// Write Own Data to CIP
      L     DB1225.DBD   10;
      T     DB1225.DBD  154;

      L     DB1225.DBW   14;
      T     DB1225.DBW  158;

      L     DB1225.DBW   16;
      T     DB1225.DBW  160;

      L     DB1225.DBW   18;
      T     DB1225.DBW  162;

      L     DB1225.DBW   20;
      T     DB1225.DBW  164;

      L     DB1225.DBW   22;
      T     DB1225.DBW  166;

      A     DB1225.DBX   24.0;
      =     DB1225.DBX  168.0;

      A     DB1225.DBX   24.1;
      =     DB1225.DBX  168.1;

      A     DB1225.DBX   24.2;
      =     DB1225.DBX  168.2;

      A     DB1225.DBX   24.3;
      =     DB1225.DBX  168.3;

      A     DB1225.DBX   24.4;
      =     DB1225.DBX  168.4;

      A     DB1225.DBX   24.5;
      =     DB1225.DBX  168.5;

      A     DB1225.DBX   24.6;
      =     DB1225.DBX  168.6;

      A     DB1225.DBX   24.7;
      =     DB1225.DBX  168.7;

// Copy Data to CIP
      CALL SFC   20 (
           SRCBLK                   := DB1225.ToCIP,
           RET_VAL                  := #iRetVal,
           DSTBLK                   := DB1225.ToCIP);

NCIP: NOP   0;

//Empty Signal
//A     "U022SpID".SpI.Sig //!!!! Insert correct Empty Signal !!!
      CLR   ;
      =     DB1225.DBX   26.5;

//Full Signal
//A     "U022SpID".SpI.Sig //!!!! Insert correct Full Signal !!!
      CLR   ;
      =     DB1225.DBX   26.2;

//CIP Program Selected
      A     #CIP;
      =     DB1225.DBX   27.1;

// Emergency Stop
      A     #EStopOK; //If needed add or replace with own SpI
      =     DB1225.DBX   27.0; //Emergency Stop OK


NETWORK
TITLE = read from other unit data



END_FUNCTION_BLOCK

FUNCTION_BLOCK FB 1229
TITLE =U022: Well Transfer VE2
AUTHOR : Woermann
FAMILY : BOTEC_F1
NAME : Sim
VERSION : 0.1


VAR_TEMP
  CIP : BOOL ;	//CIP active
  xTmp : BOOL ;	//Temporary BOOL (free for general use)
  iTmp : INT ;	//Temporary INT (free for general use)
  rTmp : REAL ;	//Temporary REAL (free for general use)
  UnitNo : INT ;	//Unit Number
END_VAR
BEGIN
NETWORK
TITLE =General

      SET   ;
// get unit number ----------------------------------------------------------
      L     DB1220.DBW    0;
      T     #UnitNo;

// CIP ----------------------------------------------------------------------
      L     DB1221.DBD   54;
      L     0;
      <D    ;
      =     #CIP;

NETWORK
TITLE =Actuator

      A     DB1221.DBX   17.3;
      =     DB2220.DBX  105.3;
      =     DB2220.DBX  185.3;
      =     DB2220.DBX  265.3;

NETWORK
TITLE =Special Input

      A     DB1221.DBX   17.3;
      =     DB2221.DBX   81.3;
      =     DB2221.DBX  141.3;
      =     DB2221.DBX  201.3;

NETWORK
TITLE =Counter

      A     DB1221.DBX   17.3;
      A     M    101.0;


      CLR   ;
NETWORK
TITLE =Analog Input

      A     DB1221.DBX   17.3;
      =     DB2223.DBX  141.3;
      =     DB2223.DBX  261.3;
      =     DB2223.DBX  381.3;

NETWORK
TITLE =Universal Value

      A     DB1221.DBX   17.3;
//      =     "U022UnVD".unv001.Sim;
//      =     "U022UnVD".unv002.Sim;
//      =     "U022UnVD".unv003.Sim;
//      =     "U022UnVD".unv004.Sim;

NETWORK
TITLE =PID

      A     DB1221.DBX   17.3;
//      =     "U022PIDD".U22_PID001.Ign;

NETWORK
TITLE =Message

      A     DB1221.DBX   17.3;
//      =     "U022MsgD".msg001.Sim;
//      =     "U022MsgD".msg002.Sim;
//      =     "U022MsgD".msg003.Sim;

NETWORK
TITLE =VLT

      A     DB1221.DBX   17.3;

END_FUNCTION_BLOCK

FUNCTION_BLOCK FB 1255
TITLE =U025: Well Transfer A
FAMILY : BOTEC_F1
NAME : Comm
VERSION : 0.1


VAR_TEMP
  iRetVal : INT ;	//return value as integer
  wRetVal : WORD ;	//return value as word
  Run : BOOL ;	//Unit in "RUN" mode
  EStopOK : BOOL ;	//Emergency Stop OK
  CIP : BOOL ;	//CIP Program Selected
  ComCIP : BOOL ;	//Communication with CIP Active
  xTmp : BOOL ;	//Temporary BOOL (free for general use)
  iTmp : INT ;	//Temporary INT (free for general use)
  rTmp : REAL ;	//Temporary REAL (free for general use)
  dTmp : DINT ;	//Temporary DINT (free for general use)
  UnitNo : INT ;	//Unit Number
  EquipmentID : INT ;	//Equipment ID
  Prid : DINT ;	//Process ID
  SFM36 : STRUCT 	// CIP Pump Mode
   I00 : BOOL ;	// Off
   I01 : BOOL ;	// Flow
   I02 : BOOL ;	// Pressure
   I03 : BOOL ;	// Fix Speed
   I04 : BOOL ;
   I05 : BOOL ;
   I06 : BOOL ;
   I07 : BOOL ;
   I08 : BOOL ;
   I09 : BOOL ;
   I10 : BOOL ;
   I11 : BOOL ;
   I12 : BOOL ;
   I13 : BOOL ;
   I14 : BOOL ;
   I15 : BOOL ;
   I16 : BOOL ;
   I17 : BOOL ;
   I18 : BOOL ;
   I19 : BOOL ;
   I20 : BOOL ;
   I21 : BOOL ;
   I22 : BOOL ;
   I23 : BOOL ;
   I24 : BOOL ;
   I25 : BOOL ;
   I26 : BOOL ;
   I27 : BOOL ;
   I28 : BOOL ;
   I29 : BOOL ;
   I30 : BOOL ;
   I31 : BOOL ;
  END_STRUCT ;
END_VAR
BEGIN
NETWORK
TITLE =general

      SET   ;

// unit & equipment number ---------------------------------------------------
      L     DB1250.DBW    0;
      T     #UnitNo;

      L     DB1255.DBW   14;
      L     1000;
      *I    ;
      L     #UnitNo;
      +I    ;
      T     #EquipmentID;

// CIP ----------------------------------------------------------------------
      L     DB1255.DBW   18;
      L     0;
      <I    ;
      =     #CIP;

// Communicating Units-------------------------------------------------------
      L     DB1255.DBD   10;
      L     DB1255.DBD  106;
      ==D   ;
      =     #ComCIP;

// emergency OK -------------------------------------------------------------
      A     DB1255.DBX   75.0; //General Emergency Stop OK
      =     #EStopOK;

NETWORK
TITLE =read other unit's data

      SET   ;

// ... General Unit ----------/

      CALL FC   563 (
           ActReq                   := M    101.0,
           PLCNo                    := DB1255.DBW   14,
           SourceUnitNo             := 99,
           IsTUnit                  := FALSE,
           DstComDRec               := DB1255.GEN,
           RET_VAL                  := #wRetVal);


NETWORK
TITLE =remote start

      SET   ;
// !!! insert correct condition of unit start !!!
      A     DB1251.DBX   15.0;
      A     DB1251.DBX   17.4;
      CLR   ;
      JCN   Strt;
      L     DB1255.DBD   10;
//L        L#-1;                            // Prid negative to start on its own
      T     #Prid;

      CALL FC    48 (
           UnitNo                   := #UnitNo,
           PrId                     := #Prid,
           Run                      := DB1251.DBX   17.4,
           PrIdTransfer             := TRUE,
           Start                    := TRUE,
           RetVal                   := #wRetVal);
Strt: NOP   0;
NETWORK
TITLE =external releases

      SET   ;
      =     DB2250.DBX  106.7;
      =     DB2250.DBX  186.7;
      =     DB2250.DBX  266.7;
NETWORK
TITLE =write own unit data

      SET   ;

//-- CIP Communication ---------------------------------------
      AN    DB1251.DBX   15.0;
//      AN "U025SeqD".Seq.PO.B30 // CIP Active (Slave)
      A     #ComCIP;
      JCN   NCIP;
//Conductivity CIP Return
      L     DB1255.DBD  150;
      T     DB1251.DBD  626;

//Temperature CIP Return
      L     DB1255.DBD  146;
      T     DB1251.DBD  594;

//CIP Prerun Pump SP

      CALL FC    45 (
           SFM                      := DB1251.DBD  686,
           Indexes                  := #SFM36);


      L     0.000000e+000;
      A     #SFM36.I01;
      =     DB1255.DBX  171.7;
      JCN   pfc;
      L     DB1251.DBD  654;
pfc:  NOP   0;
      A     #SFM36.I02;
      =     DB1255.DBX  172.0;
      JCN   ppc;
      L     DB1251.DBD  670;
ppc:  NOP   0;
      A     #SFM36.I03;
      =     DB1255.DBX  171.6;
      JCN   pxc;
      L     DB1251.DBD  574;
pxc:  NOP   0;
      T     DB1255.DBD  182;

//CIP Return
      L     DB1251.DBD  558;
      T     DB1255.DBD  186;
      L     DB1255.DBD  138;
      T     DB1251.DBD  562;

//CIP Prerun
      L     DB1251.DBD  542;
      T     DB1255.DBD  190;
      L     DB1255.DBD  142;
      T     DB1251.DBD  546;

// Write Own Data to CIP
      L     DB1255.DBD   10;
      T     DB1255.DBD  154;

      L     DB1255.DBW   14;
      T     DB1255.DBW  158;

      L     DB1255.DBW   16;
      T     DB1255.DBW  160;

      L     DB1255.DBW   18;
      T     DB1255.DBW  162;

      L     DB1255.DBW   20;
      T     DB1255.DBW  164;

      L     DB1255.DBW   22;
      T     DB1255.DBW  166;

      A     DB1255.DBX   24.0;
      =     DB1255.DBX  168.0;

      A     DB1255.DBX   24.1;
      =     DB1255.DBX  168.1;

      A     DB1255.DBX   24.2;
      =     DB1255.DBX  168.2;

      A     DB1255.DBX   24.3;
      =     DB1255.DBX  168.3;

      A     DB1255.DBX   24.4;
      =     DB1255.DBX  168.4;

      A     DB1255.DBX   24.5;
      =     DB1255.DBX  168.5;

      A     DB1255.DBX   24.6;
      =     DB1255.DBX  168.6;

      A     DB1255.DBX   24.7;
      =     DB1255.DBX  168.7;

// Copy Data to CIP
      CALL SFC   20 (
           SRCBLK                   := DB1255.ToCIP,
           RET_VAL                  := #iRetVal,
           DSTBLK                   := DB1255.ToCIP);

NCIP: NOP   0;

//Empty Signal
//A     "U025SpID".SpI.Sig //!!!! Insert correct Empty Signal !!!
      CLR   ;
      =     DB1255.DBX   26.5;

//Full Signal
//A     "U025SpID".SpI.Sig //!!!! Insert correct Full Signal !!!
      CLR   ;
      =     DB1255.DBX   26.2;

//CIP Program Selected
      A     #CIP;
      =     DB1255.DBX   27.1;

// Emergency Stop
      A     #EStopOK; //If needed add or replace with own SpI
      =     DB1255.DBX   27.0; //Emergency Stop OK


NETWORK
TITLE = read from other unit data



END_FUNCTION_BLOCK

FUNCTION_BLOCK FB 1259
TITLE =U025: Well Transfer A
AUTHOR : Woermann
FAMILY : BOTEC_F1
NAME : Sim
VERSION : 0.1


VAR_TEMP
  CIP : BOOL ;	//CIP active
  xTmp : BOOL ;	//Temporary BOOL (free for general use)
  iTmp : INT ;	//Temporary INT (free for general use)
  rTmp : REAL ;	//Temporary REAL (free for general use)
  UnitNo : INT ;	//Unit Number
END_VAR
BEGIN
NETWORK
TITLE =General

      SET   ;
// get unit number ----------------------------------------------------------
      L     DB1250.DBW    0;
      T     #UnitNo;

// CIP ----------------------------------------------------------------------
      L     DB1251.DBD   54;
      L     0;
      <D    ;
      =     #CIP;

NETWORK
TITLE =Actuator

      A     DB1251.DBX   17.3;
      =     DB2250.DBX  105.3;
      =     DB2250.DBX  185.3;
      =     DB2250.DBX  265.3;

NETWORK
TITLE =Special Input

      A     DB1251.DBX   17.3;
      =     DB2251.DBX   81.3;
      =     DB2251.DBX  141.3;
      =     DB2251.DBX  201.3;

NETWORK
TITLE =Counter

      A     DB1251.DBX   17.3;
      A     M    101.0;


      CLR   ;
NETWORK
TITLE =Analog Input

      A     DB1251.DBX   17.3;
      =     DB2253.DBX  141.3;
      =     DB2253.DBX  261.3;
      =     DB2253.DBX  381.3;

NETWORK
TITLE =Universal Value

      A     DB1251.DBX   17.3;
//      =     "U025UnVD".unv001.Sim;
//      =     "U025UnVD".unv002.Sim;
//      =     "U025UnVD".unv003.Sim;
//      =     "U025UnVD".unv004.Sim;

NETWORK
TITLE =PID

      A     DB1251.DBX   17.3;
//      =     "U025PIDD".CO2ARV1.Ign;

NETWORK
TITLE =Message

      A     DB1251.DBX   17.3;
//      =     "U025MsgD".msg001.Sim;
//      =     "U025MsgD".msg002.Sim;
//      =     "U025MsgD".msg003.Sim;

NETWORK
TITLE =VLT

      A     DB1251.DBX   17.3;

END_FUNCTION_BLOCK

FUNCTION_BLOCK FB 1265
TITLE =U026: Well Transfer B
FAMILY : BOTEC_F1
NAME : Comm
VERSION : 0.1


VAR_TEMP
  iRetVal : INT ;	//return value as integer
  wRetVal : WORD ;	//return value as word
  Run : BOOL ;	//Unit in "RUN" mode
  EStopOK : BOOL ;	//Emergency Stop OK
  CIP : BOOL ;	//CIP Program Selected
  ComCIP : BOOL ;	//Communication with CIP Active
  xTmp : BOOL ;	//Temporary BOOL (free for general use)
  iTmp : INT ;	//Temporary INT (free for general use)
  rTmp : REAL ;	//Temporary REAL (free for general use)
  dTmp : DINT ;	//Temporary DINT (free for general use)
  UnitNo : INT ;	//Unit Number
  EquipmentID : INT ;	//Equipment ID
  Prid : DINT ;	//Process ID
  SFM36 : STRUCT 	// CIP Pump Mode
   I00 : BOOL ;	// Off
   I01 : BOOL ;	// Flow
   I02 : BOOL ;	// Pressure
   I03 : BOOL ;	// Fix Speed
   I04 : BOOL ;
   I05 : BOOL ;
   I06 : BOOL ;
   I07 : BOOL ;
   I08 : BOOL ;
   I09 : BOOL ;
   I10 : BOOL ;
   I11 : BOOL ;
   I12 : BOOL ;
   I13 : BOOL ;
   I14 : BOOL ;
   I15 : BOOL ;
   I16 : BOOL ;
   I17 : BOOL ;
   I18 : BOOL ;
   I19 : BOOL ;
   I20 : BOOL ;
   I21 : BOOL ;
   I22 : BOOL ;
   I23 : BOOL ;
   I24 : BOOL ;
   I25 : BOOL ;
   I26 : BOOL ;
   I27 : BOOL ;
   I28 : BOOL ;
   I29 : BOOL ;
   I30 : BOOL ;
   I31 : BOOL ;
  END_STRUCT ;
END_VAR
BEGIN
NETWORK
TITLE =general

      SET   ;

// unit & equipment number ---------------------------------------------------
      L     DB1260.DBW    0;
      T     #UnitNo;

      L     DB1265.DBW   14;
      L     1000;
      *I    ;
      L     #UnitNo;
      +I    ;
      T     #EquipmentID;

// CIP ----------------------------------------------------------------------
      L     DB1265.DBW   18;
      L     0;
      <I    ;
      =     #CIP;

// Communicating Units-------------------------------------------------------
      L     DB1265.DBD   10;
      L     DB1265.DBD  106;
      ==D   ;
      =     #ComCIP;

// emergency OK -------------------------------------------------------------
      A     DB1265.DBX   75.0; //General Emergency Stop OK
      =     #EStopOK;

NETWORK
TITLE =read other unit's data

      SET   ;

// ... General Unit ----------/

      CALL FC   563 (
           ActReq                   := M    101.0,
           PLCNo                    := DB1265.DBW   14,
           SourceUnitNo             := 99,
           IsTUnit                  := FALSE,
           DstComDRec               := DB1265.GEN,
           RET_VAL                  := #wRetVal);

NETWORK
TITLE =remote start

      SET   ;
// !!! insert correct condition of unit start !!!
      A     DB1261.DBX   15.0;
      A     DB1261.DBX   17.4;
      CLR   ;
      JCN   Strt;
      L     DB1265.DBD   10;
//L        L#-1;                            // Prid negative to start on its own
      T     #Prid;

      CALL FC    48 (
           UnitNo                   := #UnitNo,
           PrId                     := #Prid,
           Run                      := DB1261.DBX   17.4,
           PrIdTransfer             := TRUE,
           Start                    := TRUE,
           RetVal                   := #wRetVal);
Strt: NOP   0;
NETWORK
TITLE =external releases

      SET   ;
      =     DB2260.DBX  106.7;
      =     DB2260.DBX  186.7;
      =     DB2260.DBX  266.7;
NETWORK
TITLE =write own unit data

      SET   ;

//-- CIP Communication ---------------------------------------
      AN    DB1261.DBX   15.0;
//      AN "U026SeqD".Seq.PO.B30 // CIP Active (Slave)
      A     #ComCIP;
      JCN   NCIP;
//Conductivity CIP Return
      L     DB1265.DBD  150;
      T     DB1261.DBD  626;

//Temperature CIP Return
      L     DB1265.DBD  146;
      T     DB1261.DBD  594;

//CIP Prerun Pump SP

      CALL FC    45 (
           SFM                      := DB1261.DBD  686,
           Indexes                  := #SFM36);


      L     0.000000e+000;
      A     #SFM36.I01;
      =     DB1265.DBX  171.7;
      JCN   pfc;
      L     DB1261.DBD  654;
pfc:  NOP   0;
      A     #SFM36.I02;
      =     DB1265.DBX  172.0;
      JCN   ppc;
      L     DB1261.DBD  670;
ppc:  NOP   0;
      A     #SFM36.I03;
      =     DB1265.DBX  171.6;
      JCN   pxc;
      L     DB1261.DBD  574;
pxc:  NOP   0;
      T     DB1265.DBD  182;

//CIP Return
      L     DB1261.DBD  558;
      T     DB1265.DBD  186;
      L     DB1265.DBD  138;
      T     DB1261.DBD  562;

//CIP Prerun
      L     DB1261.DBD  542;
      T     DB1265.DBD  190;
      L     DB1265.DBD  142;
      T     DB1261.DBD  546;

// Write Own Data to CIP
      L     DB1265.DBD   10;
      T     DB1265.DBD  154;

      L     DB1265.DBW   14;
      T     DB1265.DBW  158;

      L     DB1265.DBW   16;
      T     DB1265.DBW  160;

      L     DB1265.DBW   18;
      T     DB1265.DBW  162;

      L     DB1265.DBW   20;
      T     DB1265.DBW  164;

      L     DB1265.DBW   22;
      T     DB1265.DBW  166;

      A     DB1265.DBX   24.0;
      =     DB1265.DBX  168.0;

      A     DB1265.DBX   24.1;
      =     DB1265.DBX  168.1;

      A     DB1265.DBX   24.2;
      =     DB1265.DBX  168.2;

      A     DB1265.DBX   24.3;
      =     DB1265.DBX  168.3;

      A     DB1265.DBX   24.4;
      =     DB1265.DBX  168.4;

      A     DB1265.DBX   24.5;
      =     DB1265.DBX  168.5;

      A     DB1265.DBX   24.6;
      =     DB1265.DBX  168.6;

      A     DB1265.DBX   24.7;
      =     DB1265.DBX  168.7;

// Copy Data to CIP
      CALL SFC   20 (
           SRCBLK                   := DB1265.ToCIP,
           RET_VAL                  := #iRetVal,
           DSTBLK                   := DB1265.ToCIP);

NCIP: NOP   0;

//Empty Signal
//A     "U026SpID".SpI.Sig //!!!! Insert correct Empty Signal !!!
      CLR   ;
      =     DB1265.DBX   26.5;

//Full Signal
//A     "U026SpID".SpI.Sig //!!!! Insert correct Full Signal !!!
      CLR   ;
      =     DB1265.DBX   26.2;

//CIP Program Selected
      A     #CIP;
      =     DB1265.DBX   27.1;

// Emergency Stop
      A     #EStopOK; //If needed add or replace with own SpI
      =     DB1265.DBX   27.0; //Emergency Stop OK


NETWORK
TITLE = read from other unit data



END_FUNCTION_BLOCK

FUNCTION_BLOCK FB 1269
TITLE =U026: Well Transfer B
AUTHOR : Woermann
FAMILY : BOTEC_F1
NAME : Sim
VERSION : 0.1


VAR_TEMP
  CIP : BOOL ;	//CIP active
  xTmp : BOOL ;	//Temporary BOOL (free for general use)
  iTmp : INT ;	//Temporary INT (free for general use)
  rTmp : REAL ;	//Temporary REAL (free for general use)
  UnitNo : INT ;	//Unit Number
END_VAR
BEGIN
NETWORK
TITLE =General

      SET   ;
// get unit number ----------------------------------------------------------
      L     DB1260.DBW    0;
      T     #UnitNo;

// CIP ----------------------------------------------------------------------
      L     DB1261.DBD   54;
      L     0;
      <D    ;
      =     #CIP;

NETWORK
TITLE =Actuator

      A     DB1261.DBX   17.3;
      =     DB2260.DBX  105.3;
      =     DB2260.DBX  185.3;
      =     DB2260.DBX  265.3;

NETWORK
TITLE =Special Input

      A     DB1261.DBX   17.3;
      =     DB2261.DBX   81.3;
      =     DB2261.DBX  141.3;
      =     DB2261.DBX  201.3;

NETWORK
TITLE =Counter

      A     DB1261.DBX   17.3;
      A     M    101.0;


      CLR   ;
NETWORK
TITLE =Analog Input

      A     DB1261.DBX   17.3;
      =     DB2263.DBX  141.3;
      =     DB2263.DBX  261.3;
      =     DB2263.DBX  381.3;

NETWORK
TITLE =Universal Value

      A     DB1261.DBX   17.3;
//      =     "U026UnVD".unv001.Sim;
//      =     "U026UnVD".unv002.Sim;
//      =     "U026UnVD".unv003.Sim;
//      =     "U026UnVD".unv004.Sim;

NETWORK
TITLE =PID

      A     DB1261.DBX   17.3;
//      =     "U026PIDD".CO2BRV1.Ign;

NETWORK
TITLE =Message

      A     DB1261.DBX   17.3;
//      =     "U026MsgD".msg001.Sim;
//      =     "U026MsgD".msg002.Sim;
//      =     "U026MsgD".msg003.Sim;

NETWORK
TITLE =VLT

      A     DB1261.DBX   17.3;

END_FUNCTION_BLOCK

FUNCTION_BLOCK FB 1275
TITLE =U027: Well Transfer CF
FAMILY : BOTEC_F1
NAME : Comm
VERSION : 0.1


VAR_TEMP
  iRetVal : INT ;	//return value as integer
  wRetVal : WORD ;	//return value as word
  Run : BOOL ;	//Unit in "RUN" mode
  EStopOK : BOOL ;	//Emergency Stop OK
  CIP : BOOL ;	//CIP Program Selected
  ComCIP : BOOL ;	//Communication with CIP Active
  xTmp : BOOL ;	//Temporary BOOL (free for general use)
  iTmp : INT ;	//Temporary INT (free for general use)
  rTmp : REAL ;	//Temporary REAL (free for general use)
  dTmp : DINT ;	//Temporary DINT (free for general use)
  UnitNo : INT ;	//Unit Number
  EquipmentID : INT ;	//Equipment ID
  Prid : DINT ;	//Process ID
  SFM36 : STRUCT 	// CIP Pump Mode
   I00 : BOOL ;	// Off
   I01 : BOOL ;	// Flow
   I02 : BOOL ;	// Pressure
   I03 : BOOL ;	// Fix Speed
   I04 : BOOL ;
   I05 : BOOL ;
   I06 : BOOL ;
   I07 : BOOL ;
   I08 : BOOL ;
   I09 : BOOL ;
   I10 : BOOL ;
   I11 : BOOL ;
   I12 : BOOL ;
   I13 : BOOL ;
   I14 : BOOL ;
   I15 : BOOL ;
   I16 : BOOL ;
   I17 : BOOL ;
   I18 : BOOL ;
   I19 : BOOL ;
   I20 : BOOL ;
   I21 : BOOL ;
   I22 : BOOL ;
   I23 : BOOL ;
   I24 : BOOL ;
   I25 : BOOL ;
   I26 : BOOL ;
   I27 : BOOL ;
   I28 : BOOL ;
   I29 : BOOL ;
   I30 : BOOL ;
   I31 : BOOL ;
  END_STRUCT ;
END_VAR
BEGIN
NETWORK
TITLE =general

      SET   ;

// unit & equipment number ---------------------------------------------------
      L     DB1270.DBW    0;
      T     #UnitNo;

      L     DB1275.DBW   14;
      L     1000;
      *I    ;
      L     #UnitNo;
      +I    ;
      T     #EquipmentID;

// CIP ----------------------------------------------------------------------
      L     DB1275.DBW   18;
      L     0;
      <I    ;
      =     #CIP;

// Communicating Units-------------------------------------------------------
      L     DB1275.DBD   10;
      L     DB1275.DBD  106;
      ==D   ;
      =     #ComCIP;

// emergency OK -------------------------------------------------------------
      A     DB1275.DBX   75.0; //General Emergency Stop OK
      =     #EStopOK;

NETWORK
TITLE =read other unit's data

      SET   ;

// ... General Unit ----------/

      CALL FC   563 (
           ActReq                   := M    101.0,
           PLCNo                    := DB1275.DBW   14,
           SourceUnitNo             := 99,
           IsTUnit                  := FALSE,
           DstComDRec               := DB1275.GEN,
           RET_VAL                  := #wRetVal);

NETWORK
TITLE =remote start

      SET   ;
// !!! insert correct condition of unit start !!!
      A     DB1271.DBX   15.0;
      A     DB1271.DBX   17.4;
      CLR   ;
      JCN   Strt;
      L     DB1275.DBD   10;
//L        L#-1;                            // Prid negative to start on its own
      T     #Prid;

      CALL FC    48 (
           UnitNo                   := #UnitNo,
           PrId                     := #Prid,
           Run                      := DB1271.DBX   17.4,
           PrIdTransfer             := TRUE,
           Start                    := TRUE,
           RetVal                   := #wRetVal);
Strt: NOP   0;
NETWORK
TITLE =external releases

      SET   ;
      =     DB2270.DBX  106.7;
      =     DB2270.DBX  186.7;
      =     DB2270.DBX  266.7;
NETWORK
TITLE =write own unit data

      SET   ;

//-- CIP Communication ---------------------------------------
      AN    DB1271.DBX   15.0;
//      AN "U027SeqD".Seq.PO.B30 // CIP Active (Slave)
      A     #ComCIP;
      JCN   NCIP;
//Conductivity CIP Return
      L     DB1275.DBD  150;
      T     DB1271.DBD  626;

//Temperature CIP Return
      L     DB1275.DBD  146;
      T     DB1271.DBD  594;

//CIP Prerun Pump SP

      CALL FC    45 (
           SFM                      := DB1271.DBD  686,
           Indexes                  := #SFM36);


      L     0.000000e+000;
      A     #SFM36.I01;
      =     DB1275.DBX  171.7;
      JCN   pfc;
      L     DB1271.DBD  654;
pfc:  NOP   0;
      A     #SFM36.I02;
      =     DB1275.DBX  172.0;
      JCN   ppc;
      L     DB1271.DBD  670;
ppc:  NOP   0;
      A     #SFM36.I03;
      =     DB1275.DBX  171.6;
      JCN   pxc;
      L     DB1271.DBD  574;
pxc:  NOP   0;
      T     DB1275.DBD  182;

//CIP Return
      L     DB1271.DBD  558;
      T     DB1275.DBD  186;
      L     DB1275.DBD  138;
      T     DB1271.DBD  562;

//CIP Prerun
      L     DB1271.DBD  542;
      T     DB1275.DBD  190;
      L     DB1275.DBD  142;
      T     DB1271.DBD  546;

// Write Own Data to CIP
      L     DB1275.DBD   10;
      T     DB1275.DBD  154;

      L     DB1275.DBW   14;
      T     DB1275.DBW  158;

      L     DB1275.DBW   16;
      T     DB1275.DBW  160;

      L     DB1275.DBW   18;
      T     DB1275.DBW  162;

      L     DB1275.DBW   20;
      T     DB1275.DBW  164;

      L     DB1275.DBW   22;
      T     DB1275.DBW  166;

      A     DB1275.DBX   24.0;
      =     DB1275.DBX  168.0;

      A     DB1275.DBX   24.1;
      =     DB1275.DBX  168.1;

      A     DB1275.DBX   24.2;
      =     DB1275.DBX  168.2;

      A     DB1275.DBX   24.3;
      =     DB1275.DBX  168.3;

      A     DB1275.DBX   24.4;
      =     DB1275.DBX  168.4;

      A     DB1275.DBX   24.5;
      =     DB1275.DBX  168.5;

      A     DB1275.DBX   24.6;
      =     DB1275.DBX  168.6;

      A     DB1275.DBX   24.7;
      =     DB1275.DBX  168.7;

// Copy Data to CIP
      CALL SFC   20 (
           SRCBLK                   := DB1275.ToCIP,
           RET_VAL                  := #iRetVal,
           DSTBLK                   := DB1275.ToCIP);

NCIP: NOP   0;

//Empty Signal
//A     "U027SpID".SpI.Sig //!!!! Insert correct Empty Signal !!!
      CLR   ;
      =     DB1275.DBX   26.5;

//Full Signal
//A     "U027SpID".SpI.Sig //!!!! Insert correct Full Signal !!!
      CLR   ;
      =     DB1275.DBX   26.2;

//CIP Program Selected
      A     #CIP;
      =     DB1275.DBX   27.1;

// Emergency Stop
      A     #EStopOK; //If needed add or replace with own SpI
      =     DB1275.DBX   27.0; //Emergency Stop OK


NETWORK
TITLE = read from other unit data



END_FUNCTION_BLOCK

FUNCTION_BLOCK FB 1279
TITLE =U027: Well Transfer CF
AUTHOR : Woermann
FAMILY : BOTEC_F1
NAME : Sim
VERSION : 0.1


VAR_TEMP
  CIP : BOOL ;	//CIP active
  xTmp : BOOL ;	//Temporary BOOL (free for general use)
  iTmp : INT ;	//Temporary INT (free for general use)
  rTmp : REAL ;	//Temporary REAL (free for general use)
  UnitNo : INT ;	//Unit Number
END_VAR
BEGIN
NETWORK
TITLE =General

      SET   ;
// get unit number ----------------------------------------------------------
      L     DB1270.DBW    0;
      T     #UnitNo;

// CIP ----------------------------------------------------------------------
      L     DB1271.DBD   54;
      L     0;
      <D    ;
      =     #CIP;

NETWORK
TITLE =Actuator

      A     DB1271.DBX   17.3;
      =     DB2270.DBX  105.3;
      =     DB2270.DBX  185.3;
      =     DB2270.DBX  265.3;

NETWORK
TITLE =Special Input

      A     DB1271.DBX   17.3;
      =     DB2271.DBX   81.3;
      =     DB2271.DBX  141.3;
      =     DB2271.DBX  201.3;

NETWORK
TITLE =Counter

      A     DB1271.DBX   17.3;
      A     M    101.0;


      CLR   ;
NETWORK
TITLE =Analog Input

      A     DB1271.DBX   17.3;
      =     DB2273.DBX  141.3;
      =     DB2273.DBX  261.3;
      =     DB2273.DBX  381.3;

NETWORK
TITLE =Universal Value

      A     DB1271.DBX   17.3;
//      =     "U027UnVD".unv001.Sim;
//      =     "U027UnVD".unv002.Sim;
//      =     "U027UnVD".unv003.Sim;
//      =     "U027UnVD".unv004.Sim;

NETWORK
TITLE =PID

      A     DB1271.DBX   17.3;
//      =     "U027PIDD".CO2CFRV1.Ign;

NETWORK
TITLE =Message

      A     DB1271.DBX   17.3;
//      =     "U027MsgD".msg001.Sim;
//      =     "U027MsgD".msg002.Sim;
//      =     "U027MsgD".msg003.Sim;

NETWORK
TITLE =VLT

      A     DB1271.DBX   17.3;

END_FUNCTION_BLOCK

FUNCTION_BLOCK FB 1285
TITLE =U028: Well Transfer C
FAMILY : BOTEC_F1
NAME : Comm
VERSION : 0.1


VAR_TEMP
  iRetVal : INT ;	//return value as integer
  wRetVal : WORD ;	//return value as word
  Run : BOOL ;	//Unit in "RUN" mode
  EStopOK : BOOL ;	//Emergency Stop OK
  CIP : BOOL ;	//CIP Program Selected
  ComCIP : BOOL ;	//Communication with CIP Active
  xTmp : BOOL ;	//Temporary BOOL (free for general use)
  iTmp : INT ;	//Temporary INT (free for general use)
  rTmp : REAL ;	//Temporary REAL (free for general use)
  dTmp : DINT ;	//Temporary DINT (free for general use)
  UnitNo : INT ;	//Unit Number
  EquipmentID : INT ;	//Equipment ID
  Prid : DINT ;	//Process ID
  SFM36 : STRUCT 	// CIP Pump Mode
   I00 : BOOL ;	// Off
   I01 : BOOL ;	// Flow
   I02 : BOOL ;	// Pressure
   I03 : BOOL ;	// Fix Speed
   I04 : BOOL ;
   I05 : BOOL ;
   I06 : BOOL ;
   I07 : BOOL ;
   I08 : BOOL ;
   I09 : BOOL ;
   I10 : BOOL ;
   I11 : BOOL ;
   I12 : BOOL ;
   I13 : BOOL ;
   I14 : BOOL ;
   I15 : BOOL ;
   I16 : BOOL ;
   I17 : BOOL ;
   I18 : BOOL ;
   I19 : BOOL ;
   I20 : BOOL ;
   I21 : BOOL ;
   I22 : BOOL ;
   I23 : BOOL ;
   I24 : BOOL ;
   I25 : BOOL ;
   I26 : BOOL ;
   I27 : BOOL ;
   I28 : BOOL ;
   I29 : BOOL ;
   I30 : BOOL ;
   I31 : BOOL ;
  END_STRUCT ;
END_VAR
BEGIN
NETWORK
TITLE =general

      SET   ;

// unit & equipment number ---------------------------------------------------
      L     DB1280.DBW    0;
      T     #UnitNo;

      L     DB1285.DBW   14;
      L     1000;
      *I    ;
      L     #UnitNo;
      +I    ;
      T     #EquipmentID;

// CIP ----------------------------------------------------------------------
      L     DB1285.DBW   18;
      L     0;
      <I    ;
      =     #CIP;

// Communicating Units-------------------------------------------------------
      L     DB1285.DBD   10;
      L     DB1285.DBD  106;
      ==D   ;
      =     #ComCIP;

// emergency OK -------------------------------------------------------------
      A     DB1285.DBX   75.0; //General Emergency Stop OK
      =     #EStopOK;

NETWORK
TITLE =read other unit's data

      SET   ;

// ... General Unit ----------/

      CALL FC   563 (
           ActReq                   := M    101.0,
           PLCNo                    := DB1285.DBW   14,
           SourceUnitNo             := 99,
           IsTUnit                  := FALSE,
           DstComDRec               := DB1285.GEN,
           RET_VAL                  := #wRetVal);

NETWORK
TITLE =remote start

      SET   ;
// !!! insert correct condition of unit start !!!
      A     DB1281.DBX   15.0;
      A     DB1281.DBX   17.4;
      CLR   ;
      JCN   Strt;
      L     DB1285.DBD   10;
//L        L#-1;                            // Prid negative to start on its own
      T     #Prid;

      CALL FC    48 (
           UnitNo                   := #UnitNo,
           PrId                     := #Prid,
           Run                      := DB1281.DBX   17.4,
           PrIdTransfer             := TRUE,
           Start                    := TRUE,
           RetVal                   := #wRetVal);
Strt: NOP   0;
NETWORK
TITLE =external releases

      SET   ;
      =     DB2280.DBX  106.7;
      =     DB2280.DBX  186.7;
      =     DB2280.DBX  266.7;
NETWORK
TITLE =write own unit data

      SET   ;

//-- CIP Communication ---------------------------------------
      AN    DB1281.DBX   15.0;
//      AN "U028SeqD".Seq.PO.B30 // CIP Active (Slave)
      A     #ComCIP;
      JCN   NCIP;
//Conductivity CIP Return
      L     DB1285.DBD  150;
      T     DB1281.DBD  626;

//Temperature CIP Return
      L     DB1285.DBD  146;
      T     DB1281.DBD  594;

//CIP Prerun Pump SP

      CALL FC    45 (
           SFM                      := DB1281.DBD  686,
           Indexes                  := #SFM36);


      L     0.000000e+000;
      A     #SFM36.I01;
      =     DB1285.DBX  171.7;
      JCN   pfc;
      L     DB1281.DBD  654;
pfc:  NOP   0;
      A     #SFM36.I02;
      =     DB1285.DBX  172.0;
      JCN   ppc;
      L     DB1281.DBD  670;
ppc:  NOP   0;
      A     #SFM36.I03;
      =     DB1285.DBX  171.6;
      JCN   pxc;
      L     DB1281.DBD  574;
pxc:  NOP   0;
      T     DB1285.DBD  182;

//CIP Return
      L     DB1281.DBD  558;
      T     DB1285.DBD  186;
      L     DB1285.DBD  138;
      T     DB1281.DBD  562;

//CIP Prerun
      L     DB1281.DBD  542;
      T     DB1285.DBD  190;
      L     DB1285.DBD  142;
      T     DB1281.DBD  546;

// Write Own Data to CIP
      L     DB1285.DBD   10;
      T     DB1285.DBD  154;

      L     DB1285.DBW   14;
      T     DB1285.DBW  158;

      L     DB1285.DBW   16;
      T     DB1285.DBW  160;

      L     DB1285.DBW   18;
      T     DB1285.DBW  162;

      L     DB1285.DBW   20;
      T     DB1285.DBW  164;

      L     DB1285.DBW   22;
      T     DB1285.DBW  166;

      A     DB1285.DBX   24.0;
      =     DB1285.DBX  168.0;

      A     DB1285.DBX   24.1;
      =     DB1285.DBX  168.1;

      A     DB1285.DBX   24.2;
      =     DB1285.DBX  168.2;

      A     DB1285.DBX   24.3;
      =     DB1285.DBX  168.3;

      A     DB1285.DBX   24.4;
      =     DB1285.DBX  168.4;

      A     DB1285.DBX   24.5;
      =     DB1285.DBX  168.5;

      A     DB1285.DBX   24.6;
      =     DB1285.DBX  168.6;

      A     DB1285.DBX   24.7;
      =     DB1285.DBX  168.7;

// Copy Data to CIP
      CALL SFC   20 (
           SRCBLK                   := DB1285.ToCIP,
           RET_VAL                  := #iRetVal,
           DSTBLK                   := DB1285.ToCIP);

NCIP: NOP   0;

//Empty Signal
//A     "U028SpID".SpI.Sig //!!!! Insert correct Empty Signal !!!
      CLR   ;
      =     DB1285.DBX   26.5;

//Full Signal
//A     "U028SpID".SpI.Sig //!!!! Insert correct Full Signal !!!
      CLR   ;
      =     DB1285.DBX   26.2;

//CIP Program Selected
      A     #CIP;
      =     DB1285.DBX   27.1;

// Emergency Stop
      A     #EStopOK; //If needed add or replace with own SpI
      =     DB1285.DBX   27.0; //Emergency Stop OK


NETWORK
TITLE = read from other unit data



END_FUNCTION_BLOCK

FUNCTION_BLOCK FB 1289
TITLE =U028: Well Transfer C
AUTHOR : Woermann
FAMILY : BOTEC_F1
NAME : Sim
VERSION : 0.1


VAR_TEMP
  CIP : BOOL ;	//CIP active
  xTmp : BOOL ;	//Temporary BOOL (free for general use)
  iTmp : INT ;	//Temporary INT (free for general use)
  rTmp : REAL ;	//Temporary REAL (free for general use)
  UnitNo : INT ;	//Unit Number
END_VAR
BEGIN
NETWORK
TITLE =General

      SET   ;
// get unit number ----------------------------------------------------------
      L     DB1280.DBW    0;
      T     #UnitNo;

// CIP ----------------------------------------------------------------------
      L     DB1281.DBD   54;
      L     0;
      <D    ;
      =     #CIP;

NETWORK
TITLE =Actuator

      A     DB1281.DBX   17.3;
      =     DB2280.DBX  105.3;
      =     DB2280.DBX  185.3;
      =     DB2280.DBX  265.3;

NETWORK
TITLE =Special Input

      A     DB1281.DBX   17.3;
      =     DB2281.DBX   81.3;
      =     DB2281.DBX  141.3;
      =     DB2281.DBX  201.3;

NETWORK
TITLE =Counter

      A     DB1281.DBX   17.3;
      A     M    101.0;


      CLR   ;
NETWORK
TITLE =Analog Input

      A     DB1281.DBX   17.3;
      =     DB2283.DBX  141.3;
      =     DB2283.DBX  261.3;
      =     DB2283.DBX  381.3;

NETWORK
TITLE =Universal Value

      A     DB1281.DBX   17.3;
//      =     "U028UnVD".unv001.Sim;
//      =     "U028UnVD".unv002.Sim;
//      =     "U028UnVD".unv003.Sim;
//      =     "U028UnVD".unv004.Sim;

NETWORK
TITLE =PID

      A     DB1281.DBX   17.3;
//      =     "U028PIDD".CO2CRV1.Ign;

NETWORK
TITLE =Message

      A     DB1281.DBX   17.3;
//      =     "U028MsgD".msg001.Sim;
//      =     "U028MsgD".msg002.Sim;
//      =     "U028MsgD".msg003.Sim;

NETWORK
TITLE =VLT

      A     DB1281.DBX   17.3;

END_FUNCTION_BLOCK

FUNCTION_BLOCK FB 1295
TITLE =U029: Well Transfer B6F
FAMILY : BOTEC_F1
NAME : Comm
VERSION : 0.1


VAR_TEMP
  iRetVal : INT ;	//return value as integer
  wRetVal : WORD ;	//return value as word
  Run : BOOL ;	//Unit in "RUN" mode
  EStopOK : BOOL ;	//Emergency Stop OK
  CIP : BOOL ;	//CIP Program Selected
  ComCIP : BOOL ;	//Communication with CIP Active
  xTmp : BOOL ;	//Temporary BOOL (free for general use)
  iTmp : INT ;	//Temporary INT (free for general use)
  rTmp : REAL ;	//Temporary REAL (free for general use)
  dTmp : DINT ;	//Temporary DINT (free for general use)
  UnitNo : INT ;	//Unit Number
  EquipmentID : INT ;	//Equipment ID
  Prid : DINT ;	//Process ID
  SFM36 : STRUCT 	// CIP Pump Mode
   I00 : BOOL ;	// Off
   I01 : BOOL ;	// Flow
   I02 : BOOL ;	// Pressure
   I03 : BOOL ;	// Fix Speed
   I04 : BOOL ;
   I05 : BOOL ;
   I06 : BOOL ;
   I07 : BOOL ;
   I08 : BOOL ;
   I09 : BOOL ;
   I10 : BOOL ;
   I11 : BOOL ;
   I12 : BOOL ;
   I13 : BOOL ;
   I14 : BOOL ;
   I15 : BOOL ;
   I16 : BOOL ;
   I17 : BOOL ;
   I18 : BOOL ;
   I19 : BOOL ;
   I20 : BOOL ;
   I21 : BOOL ;
   I22 : BOOL ;
   I23 : BOOL ;
   I24 : BOOL ;
   I25 : BOOL ;
   I26 : BOOL ;
   I27 : BOOL ;
   I28 : BOOL ;
   I29 : BOOL ;
   I30 : BOOL ;
   I31 : BOOL ;
  END_STRUCT ;
END_VAR
BEGIN
NETWORK
TITLE =general

      SET   ;

// unit & equipment number ---------------------------------------------------
      L     DB1290.DBW    0;
      T     #UnitNo;

      L     DB1295.DBW   14;
      L     1000;
      *I    ;
      L     #UnitNo;
      +I    ;
      T     #EquipmentID;

// CIP ----------------------------------------------------------------------
      L     DB1295.DBW   18;
      L     0;
      <I    ;
      =     #CIP;

// Communicating Units-------------------------------------------------------
      L     DB1295.DBD   10;
      L     DB1295.DBD  106;
      ==D   ;
      =     #ComCIP;

// emergency OK -------------------------------------------------------------
      A     DB1295.DBX   75.0; //General Emergency Stop OK
      =     #EStopOK;

NETWORK
TITLE =read other unit's data

      SET   ;

// ... General Unit ----------/

      CALL FC   563 (
           ActReq                   := M    101.0,
           PLCNo                    := DB1295.DBW   14,
           SourceUnitNo             := 99,
           IsTUnit                  := FALSE,
           DstComDRec               := DB1295.GEN,
           RET_VAL                  := #wRetVal);


NETWORK
TITLE =remote start

      SET   ;
// !!! insert correct condition of unit start !!!
      A     DB1291.DBX   15.0;
      A     DB1291.DBX   17.4;
      CLR   ;
      JCN   Strt;
      L     DB1295.DBD   10;
//L        L#-1;                            // Prid negative to start on its own
      T     #Prid;

      CALL FC    48 (
           UnitNo                   := #UnitNo,
           PrId                     := #Prid,
           Run                      := DB1291.DBX   17.4,
           PrIdTransfer             := TRUE,
           Start                    := TRUE,
           RetVal                   := #wRetVal);
Strt: NOP   0;
NETWORK
TITLE =external releases

      SET   ;
      =     DB2290.DBX  106.7;
      =     DB2290.DBX  186.7;
      =     DB2290.DBX  266.7;
NETWORK
TITLE =write own unit data

      SET   ;

//-- CIP Communication ---------------------------------------
      AN    DB1291.DBX   15.0;
//      AN "U029SeqD".Seq.PO.B30 // CIP Active (Slave)
      A     #ComCIP;
      JCN   NCIP;
//Conductivity CIP Return
      L     DB1295.DBD  150;
      T     DB1291.DBD  626;

//Temperature CIP Return
      L     DB1295.DBD  146;
      T     DB1291.DBD  594;

//CIP Prerun Pump SP

      CALL FC    45 (
           SFM                      := DB1291.DBD  686,
           Indexes                  := #SFM36);


      L     0.000000e+000;
      A     #SFM36.I01;
      =     DB1295.DBX  171.7;
      JCN   pfc;
      L     DB1291.DBD  654;
pfc:  NOP   0;
      A     #SFM36.I02;
      =     DB1295.DBX  172.0;
      JCN   ppc;
      L     DB1291.DBD  670;
ppc:  NOP   0;
      A     #SFM36.I03;
      =     DB1295.DBX  171.6;
      JCN   pxc;
      L     DB1291.DBD  574;
pxc:  NOP   0;
      T     DB1295.DBD  182;

//CIP Return
      L     DB1291.DBD  558;
      T     DB1295.DBD  186;
      L     DB1295.DBD  138;
      T     DB1291.DBD  562;

//CIP Prerun
      L     DB1291.DBD  542;
      T     DB1295.DBD  190;
      L     DB1295.DBD  142;
      T     DB1291.DBD  546;

// Write Own Data to CIP
      L     DB1295.DBD   10;
      T     DB1295.DBD  154;

      L     DB1295.DBW   14;
      T     DB1295.DBW  158;

      L     DB1295.DBW   16;
      T     DB1295.DBW  160;

      L     DB1295.DBW   18;
      T     DB1295.DBW  162;

      L     DB1295.DBW   20;
      T     DB1295.DBW  164;

      L     DB1295.DBW   22;
      T     DB1295.DBW  166;

      A     DB1295.DBX   24.0;
      =     DB1295.DBX  168.0;

      A     DB1295.DBX   24.1;
      =     DB1295.DBX  168.1;

      A     DB1295.DBX   24.2;
      =     DB1295.DBX  168.2;

      A     DB1295.DBX   24.3;
      =     DB1295.DBX  168.3;

      A     DB1295.DBX   24.4;
      =     DB1295.DBX  168.4;

      A     DB1295.DBX   24.5;
      =     DB1295.DBX  168.5;

      A     DB1295.DBX   24.6;
      =     DB1295.DBX  168.6;

      A     DB1295.DBX   24.7;
      =     DB1295.DBX  168.7;

// Copy Data to CIP
      CALL SFC   20 (
           SRCBLK                   := DB1295.ToCIP,
           RET_VAL                  := #iRetVal,
           DSTBLK                   := DB1295.ToCIP);

NCIP: NOP   0;

//Empty Signal
//A     "U029SpID".SpI.Sig //!!!! Insert correct Empty Signal !!!
      CLR   ;
      =     DB1295.DBX   26.5;

//Full Signal
//A     "U029SpID".SpI.Sig //!!!! Insert correct Full Signal !!!
      CLR   ;
      =     DB1295.DBX   26.2;

//CIP Program Selected
      A     #CIP;
      =     DB1295.DBX   27.1;

// Emergency Stop
      A     #EStopOK; //If needed add or replace with own SpI
      =     DB1295.DBX   27.0; //Emergency Stop OK


NETWORK
TITLE = read from other unit data



END_FUNCTION_BLOCK

FUNCTION_BLOCK FB 1299
TITLE =U029: Well Transfer B6F
AUTHOR : Woermann
FAMILY : BOTEC_F1
NAME : Sim
VERSION : 0.1


VAR_TEMP
  CIP : BOOL ;	//CIP active
  xTmp : BOOL ;	//Temporary BOOL (free for general use)
  iTmp : INT ;	//Temporary INT (free for general use)
  rTmp : REAL ;	//Temporary REAL (free for general use)
  UnitNo : INT ;	//Unit Number
END_VAR
BEGIN
NETWORK
TITLE =General

      SET   ;
// get unit number ----------------------------------------------------------
      L     DB1290.DBW    0;
      T     #UnitNo;

// CIP ----------------------------------------------------------------------
      L     DB1291.DBD   54;
      L     0;
      <D    ;
      =     #CIP;

NETWORK
TITLE =Actuator

      A     DB1291.DBX   17.3;
      =     DB2290.DBX  105.3;
      =     DB2290.DBX  185.3;
      =     DB2290.DBX  265.3;

NETWORK
TITLE =Special Input

      A     DB1291.DBX   17.3;
      =     DB2291.DBX   81.3;
      =     DB2291.DBX  141.3;
      =     DB2291.DBX  201.3;

NETWORK
TITLE =Counter

      A     DB1291.DBX   17.3;
      A     M    101.0;


      CLR   ;
NETWORK
TITLE =Analog Input

      A     DB1291.DBX   17.3;
      =     DB2293.DBX  141.3;
      =     DB2293.DBX  261.3;
      =     DB2293.DBX  381.3;

NETWORK
TITLE =Universal Value

      A     DB1291.DBX   17.3;
//      =     "U029UnVD".unv001.Sim;
//      =     "U029UnVD".unv002.Sim;
//      =     "U029UnVD".unv003.Sim;
//      =     "U029UnVD".unv004.Sim;

NETWORK
TITLE =PID

      A     DB1291.DBX   17.3;
//      =     "U029PIDD".CO2B6FRV1.Ign;

NETWORK
TITLE =Message

      A     DB1291.DBX   17.3;
//      =     "U029MsgD".msg001.Sim;
//      =     "U029MsgD".msg002.Sim;
//      =     "U029MsgD".msg003.Sim;

NETWORK
TITLE =VLT

      A     DB1291.DBX   17.3;

END_FUNCTION_BLOCK

FUNCTION_BLOCK FB 1305
TITLE =U030: Well Transfer H6
FAMILY : BOTEC_F1
NAME : Comm
VERSION : 0.1


VAR_TEMP
  iRetVal : INT ;	//return value as integer
  wRetVal : WORD ;	//return value as word
  Run : BOOL ;	//Unit in "RUN" mode
  EStopOK : BOOL ;	//Emergency Stop OK
  CIP : BOOL ;	//CIP Program Selected
  ComCIP : BOOL ;	//Communication with CIP Active
  xTmp : BOOL ;	//Temporary BOOL (free for general use)
  iTmp : INT ;	//Temporary INT (free for general use)
  rTmp : REAL ;	//Temporary REAL (free for general use)
  dTmp : DINT ;	//Temporary DINT (free for general use)
  UnitNo : INT ;	//Unit Number
  EquipmentID : INT ;	//Equipment ID
  Prid : DINT ;	//Process ID
  SFM36 : STRUCT 	// CIP Pump Mode
   I00 : BOOL ;	// Off
   I01 : BOOL ;	// Flow
   I02 : BOOL ;	// Pressure
   I03 : BOOL ;	// Fix Speed
   I04 : BOOL ;
   I05 : BOOL ;
   I06 : BOOL ;
   I07 : BOOL ;
   I08 : BOOL ;
   I09 : BOOL ;
   I10 : BOOL ;
   I11 : BOOL ;
   I12 : BOOL ;
   I13 : BOOL ;
   I14 : BOOL ;
   I15 : BOOL ;
   I16 : BOOL ;
   I17 : BOOL ;
   I18 : BOOL ;
   I19 : BOOL ;
   I20 : BOOL ;
   I21 : BOOL ;
   I22 : BOOL ;
   I23 : BOOL ;
   I24 : BOOL ;
   I25 : BOOL ;
   I26 : BOOL ;
   I27 : BOOL ;
   I28 : BOOL ;
   I29 : BOOL ;
   I30 : BOOL ;
   I31 : BOOL ;
  END_STRUCT ;
END_VAR
BEGIN
NETWORK
TITLE =general

      SET   ;

// unit & equipment number ---------------------------------------------------
      L     DB1300.DBW    0;
      T     #UnitNo;

      L     DB1305.DBW   14;
      L     1000;
      *I    ;
      L     #UnitNo;
      +I    ;
      T     #EquipmentID;

// CIP ----------------------------------------------------------------------
      L     DB1305.DBW   18;
      L     0;
      <I    ;
      =     #CIP;

// Communicating Units-------------------------------------------------------
      L     DB1305.DBD   10;
      L     DB1305.DBD  106;
      ==D   ;
      =     #ComCIP;

// emergency OK -------------------------------------------------------------
      A     DB1305.DBX   75.0; //General Emergency Stop OK
      =     #EStopOK;

NETWORK
TITLE =read other unit's data

      SET   ;

// ... General Unit ----------/

      CALL FC   563 (
           ActReq                   := M    101.0,
           PLCNo                    := DB1305.DBW   14,
           SourceUnitNo             := 99,
           IsTUnit                  := FALSE,
           DstComDRec               := DB1305.GEN,
           RET_VAL                  := #wRetVal);

NETWORK
TITLE =remote start

      SET   ;
// !!! insert correct condition of unit start !!!
      A     DB1301.DBX   15.0;
      A     DB1301.DBX   17.4;
      CLR   ;
      JCN   Strt;
      L     DB1305.DBD   10;
//L        L#-1;                            // Prid negative to start on its own
      T     #Prid;

      CALL FC    48 (
           UnitNo                   := #UnitNo,
           PrId                     := #Prid,
           Run                      := DB1301.DBX   17.4,
           PrIdTransfer             := TRUE,
           Start                    := TRUE,
           RetVal                   := #wRetVal);
Strt: NOP   0;
NETWORK
TITLE =external releases

      SET   ;
      =     DB2300.DBX  106.7;
      =     DB2300.DBX  186.7;
      =     DB2300.DBX  266.7;
NETWORK
TITLE =write own unit data

      SET   ;

//-- CIP Communication ---------------------------------------
      AN    DB1301.DBX   15.0;
//      AN "U030SeqD".Seq.PO.B30 // CIP Active (Slave)
      A     #ComCIP;
      JCN   NCIP;
//Conductivity CIP Return
      L     DB1305.DBD  150;
      T     DB1301.DBD  626;

//Temperature CIP Return
      L     DB1305.DBD  146;
      T     DB1301.DBD  594;

//CIP Prerun Pump SP

      CALL FC    45 (
           SFM                      := DB1301.DBD  686,
           Indexes                  := #SFM36);


      L     0.000000e+000;
      A     #SFM36.I01;
      =     DB1305.DBX  171.7;
      JCN   pfc;
      L     DB1301.DBD  654;
pfc:  NOP   0;
      A     #SFM36.I02;
      =     DB1305.DBX  172.0;
      JCN   ppc;
      L     DB1301.DBD  670;
ppc:  NOP   0;
      A     #SFM36.I03;
      =     DB1305.DBX  171.6;
      JCN   pxc;
      L     DB1301.DBD  574;
pxc:  NOP   0;
      T     DB1305.DBD  182;

//CIP Return
      L     DB1301.DBD  558;
      T     DB1305.DBD  186;
      L     DB1305.DBD  138;
      T     DB1301.DBD  562;

//CIP Prerun
      L     DB1301.DBD  542;
      T     DB1305.DBD  190;
      L     DB1305.DBD  142;
      T     DB1301.DBD  546;

// Write Own Data to CIP
      L     DB1305.DBD   10;
      T     DB1305.DBD  154;

      L     DB1305.DBW   14;
      T     DB1305.DBW  158;

      L     DB1305.DBW   16;
      T     DB1305.DBW  160;

      L     DB1305.DBW   18;
      T     DB1305.DBW  162;

      L     DB1305.DBW   20;
      T     DB1305.DBW  164;

      L     DB1305.DBW   22;
      T     DB1305.DBW  166;

      A     DB1305.DBX   24.0;
      =     DB1305.DBX  168.0;

      A     DB1305.DBX   24.1;
      =     DB1305.DBX  168.1;

      A     DB1305.DBX   24.2;
      =     DB1305.DBX  168.2;

      A     DB1305.DBX   24.3;
      =     DB1305.DBX  168.3;

      A     DB1305.DBX   24.4;
      =     DB1305.DBX  168.4;

      A     DB1305.DBX   24.5;
      =     DB1305.DBX  168.5;

      A     DB1305.DBX   24.6;
      =     DB1305.DBX  168.6;

      A     DB1305.DBX   24.7;
      =     DB1305.DBX  168.7;

// Copy Data to CIP
      CALL SFC   20 (
           SRCBLK                   := DB1305.ToCIP,
           RET_VAL                  := #iRetVal,
           DSTBLK                   := DB1305.ToCIP);

NCIP: NOP   0;

//Empty Signal
//A     "U030SpID".SpI.Sig //!!!! Insert correct Empty Signal !!!
      CLR   ;
      =     DB1305.DBX   26.5;

//Full Signal
//A     "U030SpID".SpI.Sig //!!!! Insert correct Full Signal !!!
      CLR   ;
      =     DB1305.DBX   26.2;

//CIP Program Selected
      A     #CIP;
      =     DB1305.DBX   27.1;

// Emergency Stop
      A     #EStopOK; //If needed add or replace with own SpI
      =     DB1305.DBX   27.0; //Emergency Stop OK


NETWORK
TITLE = read from other unit data



END_FUNCTION_BLOCK

FUNCTION_BLOCK FB 1309
TITLE =U030: Well Transfer H6
AUTHOR : Woermann
FAMILY : BOTEC_F1
NAME : Sim
VERSION : 0.1


VAR_TEMP
  CIP : BOOL ;	//CIP active
  xTmp : BOOL ;	//Temporary BOOL (free for general use)
  iTmp : INT ;	//Temporary INT (free for general use)
  rTmp : REAL ;	//Temporary REAL (free for general use)
  UnitNo : INT ;	//Unit Number
END_VAR
BEGIN
NETWORK
TITLE =General

      SET   ;
// get unit number ----------------------------------------------------------
      L     DB1300.DBW    0;
      T     #UnitNo;

// CIP ----------------------------------------------------------------------
      L     DB1301.DBD   54;
      L     0;
      <D    ;
      =     #CIP;

NETWORK
TITLE =Actuator

      A     DB1301.DBX   17.3;
      =     DB2300.DBX  105.3;
      =     DB2300.DBX  185.3;
      =     DB2300.DBX  265.3;

NETWORK
TITLE =Special Input

      A     DB1301.DBX   17.3;
      =     DB2301.DBX   81.3;
      =     DB2301.DBX  141.3;
      =     DB2301.DBX  201.3;

NETWORK
TITLE =Counter

      A     DB1301.DBX   17.3;
      A     M    101.0;


      CLR   ;
NETWORK
TITLE =Analog Input

      A     DB1301.DBX   17.3;
      =     DB2303.DBX  141.3;
      =     DB2303.DBX  261.3;
      =     DB2303.DBX  381.3;

NETWORK
TITLE =Universal Value

      A     DB1301.DBX   17.3;
//      =     "U030UnVD".unv001.Sim;
//      =     "U030UnVD".unv002.Sim;
//      =     "U030UnVD".unv003.Sim;
//      =     "U030UnVD".unv004.Sim;

NETWORK
TITLE =PID

      A     DB1301.DBX   17.3;
//      =     "U030PIDD".CO2H6FRV1.Ign;

NETWORK
TITLE =Message

      A     DB1301.DBX   17.3;
//      =     "U030MsgD".msg001.Sim;
//      =     "U030MsgD".msg002.Sim;
//      =     "U030MsgD".msg003.Sim;

NETWORK
TITLE =VLT

      A     DB1301.DBX   17.3;

END_FUNCTION_BLOCK

FUNCTION_BLOCK FB 1315
TITLE =U031: Well Transfer J6
FAMILY : BOTEC_F1
NAME : Comm
VERSION : 0.1


VAR_TEMP
  iRetVal : INT ;	//return value as integer
  wRetVal : WORD ;	//return value as word
  Run : BOOL ;	//Unit in "RUN" mode
  EStopOK : BOOL ;	//Emergency Stop OK
  CIP : BOOL ;	//CIP Program Selected
  ComCIP : BOOL ;	//Communication with CIP Active
  xTmp : BOOL ;	//Temporary BOOL (free for general use)
  iTmp : INT ;	//Temporary INT (free for general use)
  rTmp : REAL ;	//Temporary REAL (free for general use)
  dTmp : DINT ;	//Temporary DINT (free for general use)
  UnitNo : INT ;	//Unit Number
  EquipmentID : INT ;	//Equipment ID
  Prid : DINT ;	//Process ID
  SFM36 : STRUCT 	// CIP Pump Mode
   I00 : BOOL ;	// Off
   I01 : BOOL ;	// Flow
   I02 : BOOL ;	// Pressure
   I03 : BOOL ;	// Fix Speed
   I04 : BOOL ;
   I05 : BOOL ;
   I06 : BOOL ;
   I07 : BOOL ;
   I08 : BOOL ;
   I09 : BOOL ;
   I10 : BOOL ;
   I11 : BOOL ;
   I12 : BOOL ;
   I13 : BOOL ;
   I14 : BOOL ;
   I15 : BOOL ;
   I16 : BOOL ;
   I17 : BOOL ;
   I18 : BOOL ;
   I19 : BOOL ;
   I20 : BOOL ;
   I21 : BOOL ;
   I22 : BOOL ;
   I23 : BOOL ;
   I24 : BOOL ;
   I25 : BOOL ;
   I26 : BOOL ;
   I27 : BOOL ;
   I28 : BOOL ;
   I29 : BOOL ;
   I30 : BOOL ;
   I31 : BOOL ;
  END_STRUCT ;
  SEND_DONE : BOOL ;
  SEND_ERROR : BOOL ;
  SEND_STATUS : WORD ;
  RECV_NDR : BOOL ;
  RECV_ERROR : BOOL ;
  RECV_STATUS : WORD ;
END_VAR
BEGIN
NETWORK
TITLE =general

      SET   ;

// unit & equipment number ---------------------------------------------------
      L     DB1310.DBW    0;
      T     #UnitNo;

      L     DB1315.DBW   14;
      L     1000;
      *I    ;
      L     #UnitNo;
      +I    ;
      T     #EquipmentID;

// CIP ----------------------------------------------------------------------
      L     DB1315.DBW   18;
      L     0;
      <I    ;
      =     #CIP;

// Communicating Units-------------------------------------------------------
      L     DB1315.DBD   10;
      L     DB1315.DBD  106;
      ==D   ;
      =     #ComCIP;

// emergency OK -------------------------------------------------------------
      A     DB1315.DBX   75.0; //General Emergency Stop OK
      =     #EStopOK;

NETWORK
TITLE = read from other unit data



NETWORK
TITLE =remote start

      SET   ;
// !!! insert correct condition of unit start !!!
      A     DB1311.DBX   15.0;
      A     DB1311.DBX   17.4;
      CLR   ;
      JCN   Strt;
      L     DB1315.DBD   10;
//L        L#-1;                            // Prid negative to start on its own
      T     #Prid;

      CALL FC    48 (
           UnitNo                   := #UnitNo,
           PrId                     := #Prid,
           Run                      := DB1311.DBX   17.4,
           PrIdTransfer             := TRUE,
           Start                    := TRUE,
           RetVal                   := #wRetVal);
Strt: NOP   0;
END_FUNCTION_BLOCK

FUNCTION_BLOCK FB 1319
TITLE =U031: Well Transfer J6
AUTHOR : Woermann
FAMILY : BOTEC_F1
NAME : Sim
VERSION : 0.1


VAR_TEMP
  CIP : BOOL ;	//CIP active
  xTmp : BOOL ;	//Temporary BOOL (free for general use)
  iTmp : INT ;	//Temporary INT (free for general use)
  rTmp : REAL ;	//Temporary REAL (free for general use)
  UnitNo : INT ;	//Unit Number
END_VAR
BEGIN
NETWORK
TITLE =General

      SET   ;
// get unit number ----------------------------------------------------------
      L     DB1310.DBW    0;
      T     #UnitNo;

// CIP ----------------------------------------------------------------------
      L     DB1311.DBD   54;
      L     0;
      <D    ;
      =     #CIP;

NETWORK
TITLE =Actuator

      A     DB1311.DBX   17.3;
      =     DB2310.DBX  105.3;
      =     DB2310.DBX  185.3;
      =     DB2310.DBX  265.3;
      =     DB2310.DBX  345.3;

NETWORK
TITLE =Special Input

      A     DB1311.DBX   17.3;
      =     DB2311.DBX   81.3;
      =     DB2311.DBX  141.3;
      =     DB2311.DBX  201.3;

NETWORK
TITLE =Counter

      A     DB1311.DBX   17.3;
      A     M    101.0;


NETWORK
TITLE =Analog Input

      A     DB1311.DBX   17.3;
      =     DB2313.DBX  141.3;
      =     DB2313.DBX  261.3;
      =     DB2313.DBX  381.3;

NETWORK
TITLE =Universal Value

      A     DB1311.DBX   17.3;
//      =     "U031UnVD".unv001.Sim;
//      =     "U031UnVD".unv002.Sim;
//      =     "U031UnVD".unv003.Sim;
//      =     "U031UnVD".unv004.Sim;

NETWORK
TITLE =PID

      A     DB1311.DBX   17.3;
//  =     "U031PIDD".CO2J6FRV1.Sim

NETWORK
TITLE =Message

      A     DB1311.DBX   17.3;
//      =     "U031MsgD".msg001.Sim;
//      =     "U031MsgD".msg002.Sim;
//      =     "U031MsgD".msg003.Sim;

NETWORK
TITLE =VLT

      A     DB1311.DBX   17.3;

END_FUNCTION_BLOCK

FUNCTION_BLOCK FB 1325
TITLE =U032: Well Transfer L6F
FAMILY : BOTEC_F1
NAME : Comm
VERSION : 0.1


VAR_TEMP
  iRetVal : INT ;	//return value as integer
  wRetVal : WORD ;	//return value as word
  Run : BOOL ;	//Unit in "RUN" mode
  EStopOK : BOOL ;	//Emergency Stop OK
  CIP : BOOL ;	//CIP Program Selected
  ComCIP : BOOL ;	//Communication with CIP Active
  xTmp : BOOL ;	//Temporary BOOL (free for general use)
  iTmp : INT ;	//Temporary INT (free for general use)
  rTmp : REAL ;	//Temporary REAL (free for general use)
  dTmp : DINT ;	//Temporary DINT (free for general use)
  UnitNo : INT ;	//Unit Number
  EquipmentID : INT ;	//Equipment ID
  Prid : DINT ;	//Process ID
  SFM36 : STRUCT 	// CIP Pump Mode
   I00 : BOOL ;	// Off
   I01 : BOOL ;	// Flow
   I02 : BOOL ;	// Pressure
   I03 : BOOL ;	// Fix Speed
   I04 : BOOL ;
   I05 : BOOL ;
   I06 : BOOL ;
   I07 : BOOL ;
   I08 : BOOL ;
   I09 : BOOL ;
   I10 : BOOL ;
   I11 : BOOL ;
   I12 : BOOL ;
   I13 : BOOL ;
   I14 : BOOL ;
   I15 : BOOL ;
   I16 : BOOL ;
   I17 : BOOL ;
   I18 : BOOL ;
   I19 : BOOL ;
   I20 : BOOL ;
   I21 : BOOL ;
   I22 : BOOL ;
   I23 : BOOL ;
   I24 : BOOL ;
   I25 : BOOL ;
   I26 : BOOL ;
   I27 : BOOL ;
   I28 : BOOL ;
   I29 : BOOL ;
   I30 : BOOL ;
   I31 : BOOL ;
  END_STRUCT ;
END_VAR
BEGIN
NETWORK
TITLE =general

      SET   ;

// unit & equipment number ---------------------------------------------------
      L     DB1320.DBW    0;
      T     #UnitNo;

      L     DB1325.DBW   14;
      L     1000;
      *I    ;
      L     #UnitNo;
      +I    ;
      T     #EquipmentID;

// CIP ----------------------------------------------------------------------
      L     DB1325.DBW   18;
      L     0;
      <I    ;
      =     #CIP;

// Communicating Units-------------------------------------------------------
      L     DB1325.DBD   10;
      L     DB1325.DBD  106;
      ==D   ;
      =     #ComCIP;

// emergency OK -------------------------------------------------------------
      A     DB1325.DBX   75.0; //General Emergency Stop OK
      =     #EStopOK;

NETWORK
TITLE =read other unit's data

      SET   ;

// ... General Unit ----------/

      CALL FC   563 (
           ActReq                   := M    101.0,
           PLCNo                    := DB1325.DBW   14,
           SourceUnitNo             := 99,
           IsTUnit                  := FALSE,
           DstComDRec               := DB1325.GEN,

           RET_VAL                  := #wRetVal);

// ... CIP Unit ------------- /

      CALL FC   563 (
           ActReq                   := M    101.0,
           PLCNo                    := 1,
           SourceUnitNo             := 71,
           IsTUnit                  := FALSE,
           DstComDRec               := DB1325.CIP,

           RET_VAL                  := #wRetVal);


NETWORK
TITLE =remote start

      SET   ;
// !!! insert correct condition of unit start !!!
      A     DB1321.DBX   15.0;
      A     DB1321.DBX   17.4;
      CLR   ;
      JCN   Strt;
      L     DB1325.DBD   10;
//L        L#-1;                            // Prid negative to start on its own
      T     #Prid;

      CALL FC    48 (
           UnitNo                   := #UnitNo,
           PrId                     := #Prid,
           Run                      := DB1321.DBX   17.4,
           PrIdTransfer             := TRUE,
           Start                    := TRUE,
           RetVal                   := #wRetVal);
Strt: NOP   0;
NETWORK
TITLE =external releases

      SET   ;
      =     DB2320.DBX  106.7;
      =     DB2320.DBX  186.7;
      =     DB2320.DBX  266.7;
NETWORK
TITLE =write own unit data

      SET   ;

//-- CIP Communication ---------------------------------------
      AN    DB1321.DBX   15.0;
//      AN "U032SeqD".Seq.PO.B30 // CIP Active (Slave)
      A     #ComCIP;
      JCN   NCIP;
//Conductivity CIP Return
      L     DB1325.DBD  150;
      T     DB1321.DBD  626;

//Temperature CIP Return
      L     DB1325.DBD  146;
      T     DB1321.DBD  594;

//CIP Prerun Pump SP

      CALL FC    45 (
           SFM                      := DB1321.DBD  686,

           Indexes                  := #SFM36);

      L     0.000000e+000;
      A     #SFM36.I01;
      =     DB1325.DBX  171.7;
      JCN   pfc;
      L     DB1321.DBD  654;
pfc:  NOP   0;
      A     #SFM36.I02;
      =     DB1325.DBX  172.0;
      JCN   ppc;
      L     DB1321.DBD  670;
ppc:  NOP   0;
      A     #SFM36.I03;
      =     DB1325.DBX  171.6;
      JCN   pxc;
      L     DB1321.DBD  574;
pxc:  NOP   0;
      T     DB1325.DBD  182;

//CIP Return
      L     DB1321.DBD  558;
      T     DB1325.DBD  186;
      L     DB1325.DBD  138;
      T     DB1321.DBD  562;

//CIP Prerun
      L     DB1321.DBD  542;
      T     DB1325.DBD  190;
      L     DB1325.DBD  142;
      T     DB1321.DBD  546;

// Write Own Data to CIP
      L     DB1325.DBD   10;
      T     DB1325.DBD  154;

      L     DB1325.DBW   14;
      T     DB1325.DBW  158;

      L     DB1325.DBW   16;
      T     DB1325.DBW  160;

      L     DB1325.DBW   18;
      T     DB1325.DBW  162;

      L     DB1325.DBW   20;
      T     DB1325.DBW  164;

      L     DB1325.DBW   22;
      T     DB1325.DBW  166;

      A     DB1325.DBX   24.0;
      =     DB1325.DBX  168.0;

      A     DB1325.DBX   24.1;
      =     DB1325.DBX  168.1;

      A     DB1325.DBX   24.2;
      =     DB1325.DBX  168.2;

      A     DB1325.DBX   24.3;
      =     DB1325.DBX  168.3;

      A     DB1325.DBX   24.4;
      =     DB1325.DBX  168.4;

      A     DB1325.DBX   24.5;
      =     DB1325.DBX  168.5;

      A     DB1325.DBX   24.6;
      =     DB1325.DBX  168.6;

      A     DB1325.DBX   24.7;
      =     DB1325.DBX  168.7;

// Copy Data to CIP
      CALL SFC   20 (
           SRCBLK                   := DB1325.ToCIP,
           RET_VAL                  := #iRetVal,
           DSTBLK                   := DB1325.ToCIP);

NCIP: NOP   0;

//Empty Signal
//A     "U032SpID".SpI.Sig //!!!! Insert correct Empty Signal !!!
      CLR   ;
      =     DB1325.DBX   26.5;

//Full Signal
//A     "U032SpID".SpI.Sig //!!!! Insert correct Full Signal !!!
      CLR   ;
      =     DB1325.DBX   26.2;

//CIP Program Selected
      A     #CIP;
      =     DB1325.DBX   27.1;

// Emergency Stop
      A     #EStopOK; //If needed add or replace with own SpI
      =     DB1325.DBX   27.0; //Emergency Stop OK


NETWORK
TITLE = read from other unit data

END_FUNCTION_BLOCK

FUNCTION_BLOCK FB 1329
TITLE =U032: Well Transfer L6F
AUTHOR : Woermann
FAMILY : BOTEC_F1
NAME : Sim
VERSION : 0.1


VAR_TEMP
  CIP : BOOL ;	//CIP active
  xTmp : BOOL ;	//Temporary BOOL (free for general use)
  iTmp : INT ;	//Temporary INT (free for general use)
  rTmp : REAL ;	//Temporary REAL (free for general use)
  UnitNo : INT ;	//Unit Number
END_VAR
BEGIN
NETWORK
TITLE =General

      SET   ;
// get unit number ----------------------------------------------------------
      L     DB1320.DBW    0;
      T     #UnitNo;

// CIP ----------------------------------------------------------------------
      L     DB1321.DBD   54;
      L     0;
      <D    ;
      =     #CIP;

NETWORK
TITLE =Actuator

      A     DB1321.DBX   17.3;
      =     DB2320.DBX  105.3;
      =     DB2320.DBX  185.3;
      =     DB2320.DBX  265.3;

NETWORK
TITLE =Special Input

      A     DB1321.DBX   17.3;
      =     DB2321.DBX   81.3;
      =     DB2321.DBX  141.3;
      =     DB2321.DBX  201.3;

NETWORK
TITLE =Counter

      A     DB1321.DBX   17.3;
      A     M    101.0;


      CLR   ;
NETWORK
TITLE =Analog Input

      A     DB1321.DBX   17.3;
      =     DB2323.DBX  141.3;
      =     DB2323.DBX  261.3;
      =     DB2323.DBX  381.3;

NETWORK
TITLE =Universal Value

      A     DB1321.DBX   17.3;
//      =     "U032UnVD".unv001.Sim;
//      =     "U032UnVD".unv002.Sim;
//      =     "U032UnVD".unv003.Sim;
//      =     "U032UnVD".unv004.Sim;

NETWORK
TITLE =PID

      A     DB1321.DBX   17.3;
//      =     "U032PIDD".CO2L6FRV1.Ign;

NETWORK
TITLE =Message

      A     DB1321.DBX   17.3;
//      =     "U032MsgD".msg001.Sim;
//      =     "U032MsgD".msg002.Sim;
//      =     "U032MsgD".msg003.Sim;

NETWORK
TITLE =VLT

      A     DB1321.DBX   17.3;

END_FUNCTION_BLOCK

FUNCTION_BLOCK FB 1335
TITLE =U033: Well Transfer B6
FAMILY : BOTEC_F1
NAME : Comm
VERSION : 0.1


VAR_TEMP
  iRetVal : INT ;	//return value as integer
  wRetVal : WORD ;	//return value as word
  Run : BOOL ;	//Unit in "RUN" mode
  EStopOK : BOOL ;	//Emergency Stop OK
  CIP : BOOL ;	//CIP Program Selected
  ComCIP : BOOL ;	//Communication with CIP Active
  xTmp : BOOL ;	//Temporary BOOL (free for general use)
  iTmp : INT ;	//Temporary INT (free for general use)
  rTmp : REAL ;	//Temporary REAL (free for general use)
  dTmp : DINT ;	//Temporary DINT (free for general use)
  UnitNo : INT ;	//Unit Number
  EquipmentID : INT ;	//Equipment ID
  Prid : DINT ;	//Process ID
  SFM36 : STRUCT 	// CIP Pump Mode
   I00 : BOOL ;	// Off
   I01 : BOOL ;	// Flow
   I02 : BOOL ;	// Pressure
   I03 : BOOL ;	// Fix Speed
   I04 : BOOL ;
   I05 : BOOL ;
   I06 : BOOL ;
   I07 : BOOL ;
   I08 : BOOL ;
   I09 : BOOL ;
   I10 : BOOL ;
   I11 : BOOL ;
   I12 : BOOL ;
   I13 : BOOL ;
   I14 : BOOL ;
   I15 : BOOL ;
   I16 : BOOL ;
   I17 : BOOL ;
   I18 : BOOL ;
   I19 : BOOL ;
   I20 : BOOL ;
   I21 : BOOL ;
   I22 : BOOL ;
   I23 : BOOL ;
   I24 : BOOL ;
   I25 : BOOL ;
   I26 : BOOL ;
   I27 : BOOL ;
   I28 : BOOL ;
   I29 : BOOL ;
   I30 : BOOL ;
   I31 : BOOL ;
  END_STRUCT ;
END_VAR
BEGIN
NETWORK
TITLE =general

      SET   ;

// unit & equipment number ---------------------------------------------------
      L     DB1330.DBW    0;
      T     #UnitNo;

      L     DB1335.DBW   14;
      L     1000;
      *I    ;
      L     #UnitNo;
      +I    ;
      T     #EquipmentID;

// CIP ----------------------------------------------------------------------
      L     DB1335.DBW   18;
      L     0;
      <I    ;
      =     #CIP;

// Communicating Units-------------------------------------------------------
      L     DB1335.DBD   10;
      L     DB1335.DBD  106;
      ==D   ;
      =     #ComCIP;

// emergency OK -------------------------------------------------------------
      A     DB1335.DBX   75.0; //General Emergency Stop OK
      =     #EStopOK;

NETWORK
TITLE =read other unit's data

      SET   ;

// ... General Unit ----------/

      CALL FC   563 (
           ActReq                   := M    101.0,
           PLCNo                    := DB1335.DBW   14,
           SourceUnitNo             := 99,
           IsTUnit                  := FALSE,
           DstComDRec               := DB1335.GEN,

           RET_VAL                  := #wRetVal);

// ... CIP Unit ------------- /

      CALL FC   563 (
           ActReq                   := M    101.0,
           PLCNo                    := 1,
           SourceUnitNo             := 71,
           IsTUnit                  := FALSE,
           DstComDRec               := DB1335.CIP,

           RET_VAL                  := #wRetVal);


NETWORK
TITLE =remote start

      SET   ;
// !!! insert correct condition of unit start !!!
      A     DB1331.DBX   15.0;
      A     DB1331.DBX   17.4;
      CLR   ;
      JCN   Strt;
      L     DB1335.DBD   10;
//L        L#-1;                            // Prid negative to start on its own
      T     #Prid;

      CALL FC    48 (
           UnitNo                   := #UnitNo,
           PrId                     := #Prid,
           Run                      := DB1331.DBX   17.4,
           PrIdTransfer             := TRUE,
           Start                    := TRUE,
           RetVal                   := #wRetVal);
Strt: NOP   0;
NETWORK
TITLE =external releases

      SET   ;
      =     DB2330.DBX  106.7;
      =     DB2330.DBX  186.7;
      =     DB2330.DBX  266.7;
NETWORK
TITLE =write own unit data

      SET   ;

//-- CIP Communication ---------------------------------------
      AN    DB1331.DBX   15.0;
//      AN "U033SeqD".Seq.PO.B30 // CIP Active (Slave)
      A     #ComCIP;
      JCN   NCIP;
//Conductivity CIP Return
      L     DB1335.DBD  150;
      T     DB1331.DBD  626;

//Temperature CIP Return
      L     DB1335.DBD  146;
      T     DB1331.DBD  594;

//CIP Prerun Pump SP

      CALL FC    45 (
           SFM                      := DB1331.DBD  686,

           Indexes                  := #SFM36);

      L     0.000000e+000;
      A     #SFM36.I01;
      =     DB1335.DBX  171.7;
      JCN   pfc;
      L     DB1331.DBD  654;
pfc:  NOP   0;
      A     #SFM36.I02;
      =     DB1335.DBX  172.0;
      JCN   ppc;
      L     DB1331.DBD  670;
ppc:  NOP   0;
      A     #SFM36.I03;
      =     DB1335.DBX  171.6;
      JCN   pxc;
      L     DB1331.DBD  574;
pxc:  NOP   0;
      T     DB1335.DBD  182;

//CIP Return
      L     DB1331.DBD  558;
      T     DB1335.DBD  186;
      L     DB1335.DBD  138;
      T     DB1331.DBD  562;

//CIP Prerun
      L     DB1331.DBD  542;
      T     DB1335.DBD  190;
      L     DB1335.DBD  142;
      T     DB1331.DBD  546;

// Write Own Data to CIP
      L     DB1335.DBD   10;
      T     DB1335.DBD  154;

      L     DB1335.DBW   14;
      T     DB1335.DBW  158;

      L     DB1335.DBW   16;
      T     DB1335.DBW  160;

      L     DB1335.DBW   18;
      T     DB1335.DBW  162;

      L     DB1335.DBW   20;
      T     DB1335.DBW  164;

      L     DB1335.DBW   22;
      T     DB1335.DBW  166;

      A     DB1335.DBX   24.0;
      =     DB1335.DBX  168.0;

      A     DB1335.DBX   24.1;
      =     DB1335.DBX  168.1;

      A     DB1335.DBX   24.2;
      =     DB1335.DBX  168.2;

      A     DB1335.DBX   24.3;
      =     DB1335.DBX  168.3;

      A     DB1335.DBX   24.4;
      =     DB1335.DBX  168.4;

      A     DB1335.DBX   24.5;
      =     DB1335.DBX  168.5;

      A     DB1335.DBX   24.6;
      =     DB1335.DBX  168.6;

      A     DB1335.DBX   24.7;
      =     DB1335.DBX  168.7;

// Copy Data to CIP
      CALL SFC   20 (
           SRCBLK                   := DB1335.ToCIP,
           RET_VAL                  := #iRetVal,
           DSTBLK                   := DB1335.ToCIP);

NCIP: NOP   0;

//Empty Signal
//A     "U033SpID".SpI.Sig //!!!! Insert correct Empty Signal !!!
      CLR   ;
      =     DB1335.DBX   26.5;

//Full Signal
//A     "U033SpID".SpI.Sig //!!!! Insert correct Full Signal !!!
      CLR   ;
      =     DB1335.DBX   26.2;

//CIP Program Selected
      A     #CIP;
      =     DB1335.DBX   27.1;

// Emergency Stop
      A     #EStopOK; //If needed add or replace with own SpI
      =     DB1335.DBX   27.0; //Emergency Stop OK


NETWORK
TITLE = read from other unit data

END_FUNCTION_BLOCK

FUNCTION_BLOCK FB 1339
TITLE =U033: Well Transfer B6
AUTHOR : Woermann
FAMILY : BOTEC_F1
NAME : Sim
VERSION : 0.1


VAR_TEMP
  CIP : BOOL ;	//CIP active
  xTmp : BOOL ;	//Temporary BOOL (free for general use)
  iTmp : INT ;	//Temporary INT (free for general use)
  rTmp : REAL ;	//Temporary REAL (free for general use)
  UnitNo : INT ;	//Unit Number
END_VAR
BEGIN
NETWORK
TITLE =General

      SET   ;
// get unit number ----------------------------------------------------------
      L     DB1330.DBW    0;
      T     #UnitNo;

// CIP ----------------------------------------------------------------------
      L     DB1331.DBD   54;
      L     0;
      <D    ;
      =     #CIP;

NETWORK
TITLE =Actuator

      A     DB1331.DBX   17.3;
      =     DB2330.DBX  105.3;
      =     DB2330.DBX  185.3;
      =     DB2330.DBX  265.3;

NETWORK
TITLE =Special Input

      A     DB1331.DBX   17.3;
      =     DB2331.DBX   81.3;
      =     DB2331.DBX  141.3;
      =     DB2331.DBX  201.3;

NETWORK
TITLE =Counter

      A     DB1331.DBX   17.3;
      A     M    101.0;


      CLR   ;
NETWORK
TITLE =Analog Input

      A     DB1331.DBX   17.3;
      =     DB2333.DBX  141.3;
      =     DB2333.DBX  261.3;
      =     DB2333.DBX  381.3;

NETWORK
TITLE =Universal Value

      A     DB1331.DBX   17.3;
//      =     "U033UnVD".unv001.Sim;
//      =     "U033UnVD".unv002.Sim;
//      =     "U033UnVD".unv003.Sim;
//      =     "U033UnVD".unv004.Sim;

NETWORK
TITLE =PID

      A     DB1331.DBX   17.3;
//      =     "U033PIDD".CO2B6RV1.Ign;

NETWORK
TITLE =Message

      A     DB1331.DBX   17.3;
//      =     "U033MsgD".msg001.Sim;
//      =     "U033MsgD".msg002.Sim;
//      =     "U033MsgD".msg003.Sim;

NETWORK
TITLE =VLT

      A     DB1331.DBX   17.3;

END_FUNCTION_BLOCK

FUNCTION_BLOCK FB 1345
TITLE =U034: Well Transfer D6
FAMILY : BOTEC_F1
NAME : Comm
VERSION : 0.1


VAR_TEMP
  iRetVal : INT ;	//return value as integer
  wRetVal : WORD ;	//return value as word
  Run : BOOL ;	//Unit in "RUN" mode
  EStopOK : BOOL ;	//Emergency Stop OK
  CIP : BOOL ;	//CIP Program Selected
  ComCIP : BOOL ;	//Communication with CIP Active
  xTmp : BOOL ;	//Temporary BOOL (free for general use)
  iTmp : INT ;	//Temporary INT (free for general use)
  rTmp : REAL ;	//Temporary REAL (free for general use)
  dTmp : DINT ;	//Temporary DINT (free for general use)
  UnitNo : INT ;	//Unit Number
  EquipmentID : INT ;	//Equipment ID
  Prid : DINT ;	//Process ID
  SFM36 : STRUCT 	// CIP Pump Mode
   I00 : BOOL ;	// Off
   I01 : BOOL ;	// Flow
   I02 : BOOL ;	// Pressure
   I03 : BOOL ;	// Fix Speed
   I04 : BOOL ;
   I05 : BOOL ;
   I06 : BOOL ;
   I07 : BOOL ;
   I08 : BOOL ;
   I09 : BOOL ;
   I10 : BOOL ;
   I11 : BOOL ;
   I12 : BOOL ;
   I13 : BOOL ;
   I14 : BOOL ;
   I15 : BOOL ;
   I16 : BOOL ;
   I17 : BOOL ;
   I18 : BOOL ;
   I19 : BOOL ;
   I20 : BOOL ;
   I21 : BOOL ;
   I22 : BOOL ;
   I23 : BOOL ;
   I24 : BOOL ;
   I25 : BOOL ;
   I26 : BOOL ;
   I27 : BOOL ;
   I28 : BOOL ;
   I29 : BOOL ;
   I30 : BOOL ;
   I31 : BOOL ;
  END_STRUCT ;
END_VAR
BEGIN
NETWORK
TITLE =general

      SET   ;

// unit & equipment number ---------------------------------------------------
      L     DB1340.DBW    0;
      T     #UnitNo;

      L     DB1345.DBW   14;
      L     1000;
      *I    ;
      L     #UnitNo;
      +I    ;
      T     #EquipmentID;

// CIP ----------------------------------------------------------------------
      L     DB1345.DBW   18;
      L     0;
      <I    ;
      =     #CIP;

// Communicating Units-------------------------------------------------------
      L     DB1345.DBD   10;
      L     DB1345.DBD  106;
      ==D   ;
      =     #ComCIP;

// emergency OK -------------------------------------------------------------
      A     DB1345.DBX   75.0; //General Emergency Stop OK
      =     #EStopOK;

NETWORK
TITLE =read other unit's data

      SET   ;

// ... General Unit ----------/

      CALL FC   563 (
           ActReq                   := M    101.0,
           PLCNo                    := DB1345.DBW   14,
           SourceUnitNo             := 99,
           IsTUnit                  := FALSE,
           DstComDRec               := DB1345.GEN,

           RET_VAL                  := #wRetVal);

// ... CIP Unit ------------- /

      CALL FC   563 (
           ActReq                   := M    101.0,
           PLCNo                    := 1,
           SourceUnitNo             := 71,
           IsTUnit                  := FALSE,
           DstComDRec               := DB1345.CIP,

           RET_VAL                  := #wRetVal);


NETWORK
TITLE =remote start

      SET   ;
// !!! insert correct condition of unit start !!!
      A     DB1341.DBX   15.0;
      A     DB1341.DBX   17.4;
      CLR   ;
      JCN   Strt;
      L     DB1345.DBD   10;
//L        L#-1;                            // Prid negative to start on its own
      T     #Prid;

      CALL FC    48 (
           UnitNo                   := #UnitNo,
           PrId                     := #Prid,
           Run                      := DB1341.DBX   17.4,
           PrIdTransfer             := TRUE,
           Start                    := TRUE,
           RetVal                   := #wRetVal);
Strt: NOP   0;
NETWORK
TITLE =external releases

      SET   ;
      =     DB2340.DBX  106.7;
      =     DB2340.DBX  186.7;
      =     DB2340.DBX  266.7;
NETWORK
TITLE =write own unit data

      SET   ;

//-- CIP Communication ---------------------------------------
      AN    DB1341.DBX   15.0;
//      AN "U034SeqD".Seq.PO.B30 // CIP Active (Slave)
      A     #ComCIP;
      JCN   NCIP;
//Conductivity CIP Return
      L     DB1345.DBD  150;
      T     DB1341.DBD  626;

//Temperature CIP Return
      L     DB1345.DBD  146;
      T     DB1341.DBD  594;

//CIP Prerun Pump SP

      CALL FC    45 (
           SFM                      := DB1341.DBD  686,

           Indexes                  := #SFM36);

      L     0.000000e+000;
      A     #SFM36.I01;
      =     DB1345.DBX  171.7;
      JCN   pfc;
      L     DB1341.DBD  654;
pfc:  NOP   0;
      A     #SFM36.I02;
      =     DB1345.DBX  172.0;
      JCN   ppc;
      L     DB1341.DBD  670;
ppc:  NOP   0;
      A     #SFM36.I03;
      =     DB1345.DBX  171.6;
      JCN   pxc;
      L     DB1341.DBD  574;
pxc:  NOP   0;
      T     DB1345.DBD  182;

//CIP Return
      L     DB1341.DBD  558;
      T     DB1345.DBD  186;
      L     DB1345.DBD  138;
      T     DB1341.DBD  562;

//CIP Prerun
      L     DB1341.DBD  542;
      T     DB1345.DBD  190;
      L     DB1345.DBD  142;
      T     DB1341.DBD  546;

// Write Own Data to CIP
      L     DB1345.DBD   10;
      T     DB1345.DBD  154;

      L     DB1345.DBW   14;
      T     DB1345.DBW  158;

      L     DB1345.DBW   16;
      T     DB1345.DBW  160;

      L     DB1345.DBW   18;
      T     DB1345.DBW  162;

      L     DB1345.DBW   20;
      T     DB1345.DBW  164;

      L     DB1345.DBW   22;
      T     DB1345.DBW  166;

      A     DB1345.DBX   24.0;
      =     DB1345.DBX  168.0;

      A     DB1345.DBX   24.1;
      =     DB1345.DBX  168.1;

      A     DB1345.DBX   24.2;
      =     DB1345.DBX  168.2;

      A     DB1345.DBX   24.3;
      =     DB1345.DBX  168.3;

      A     DB1345.DBX   24.4;
      =     DB1345.DBX  168.4;

      A     DB1345.DBX   24.5;
      =     DB1345.DBX  168.5;

      A     DB1345.DBX   24.6;
      =     DB1345.DBX  168.6;

      A     DB1345.DBX   24.7;
      =     DB1345.DBX  168.7;

// Copy Data to CIP
      CALL SFC   20 (
           SRCBLK                   := DB1345.ToCIP,
           RET_VAL                  := #iRetVal,
           DSTBLK                   := DB1345.ToCIP);

NCIP: NOP   0;

//Empty Signal
//A     "U034SpID".SpI.Sig //!!!! Insert correct Empty Signal !!!
      CLR   ;
      =     DB1345.DBX   26.5;

//Full Signal
//A     "U034SpID".SpI.Sig //!!!! Insert correct Full Signal !!!
      CLR   ;
      =     DB1345.DBX   26.2;

//CIP Program Selected
      A     #CIP;
      =     DB1345.DBX   27.1;

// Emergency Stop
      A     #EStopOK; //If needed add or replace with own SpI
      =     DB1345.DBX   27.0; //Emergency Stop OK


NETWORK
TITLE = read from other unit data

END_FUNCTION_BLOCK

FUNCTION_BLOCK FB 1349
TITLE =U034: Well Transfer D6
AUTHOR : Woermann
FAMILY : BOTEC_F1
NAME : Sim
VERSION : 0.1


VAR_TEMP
  CIP : BOOL ;	//CIP active
  xTmp : BOOL ;	//Temporary BOOL (free for general use)
  iTmp : INT ;	//Temporary INT (free for general use)
  rTmp : REAL ;	//Temporary REAL (free for general use)
  UnitNo : INT ;	//Unit Number
END_VAR
BEGIN
NETWORK
TITLE =General

      SET   ;
// get unit number ----------------------------------------------------------
      L     DB1340.DBW    0;
      T     #UnitNo;

// CIP ----------------------------------------------------------------------
      L     DB1341.DBD   54;
      L     0;
      <D    ;
      =     #CIP;

NETWORK
TITLE =Actuator

      A     DB1341.DBX   17.3;
      =     DB2340.DBX  105.3;
      =     DB2340.DBX  185.3;
      =     DB2340.DBX  265.3;

NETWORK
TITLE =Special Input

      A     DB1341.DBX   17.3;
      =     DB2341.DBX   81.3;
      =     DB2341.DBX  141.3;
      =     DB2341.DBX  201.3;

NETWORK
TITLE =Counter

      A     DB1341.DBX   17.3;
      A     M    101.0;


      CLR   ;
NETWORK
TITLE =Analog Input

      A     DB1341.DBX   17.3;
      =     DB2343.DBX  141.3;
      =     DB2343.DBX  261.3;
      =     DB2343.DBX  381.3;

NETWORK
TITLE =Universal Value

      A     DB1341.DBX   17.3;
//      =     "U034UnVD".unv001.Sim;
//      =     "U034UnVD".unv002.Sim;
//      =     "U034UnVD".unv003.Sim;
//      =     "U034UnVD".unv004.Sim;

NETWORK
TITLE =PID

      A     DB1341.DBX   17.3;
//      =     "U034PIDD".CO2D6RV1.Ign;

NETWORK
TITLE =Message

      A     DB1341.DBX   17.3;
//      =     "U034MsgD".msg001.Sim;
//      =     "U034MsgD".msg002.Sim;
//      =     "U034MsgD".msg003.Sim;

NETWORK
TITLE =VLT

      A     DB1341.DBX   17.3;

END_FUNCTION_BLOCK

FUNCTION_BLOCK FB 1385
TITLE =U038: Water Treatment 1
FAMILY : BOTEC_F1
NAME : Comm
VERSION : 0.1


VAR_TEMP
  iRetVal : INT ;	//return value as integer
  wRetVal : WORD ;	//return value as word
  Run : BOOL ;	//Unit in "RUN" mode
  EStopOK : BOOL ;	//Emergency Stop OK
  CIP : BOOL ;	//CIP Program Selected
  ComCIP : BOOL ;	//Communication with CIP Active
  xTmp : BOOL ;	//Temporary BOOL (free for general use)
  iTmp : INT ;	//Temporary INT (free for general use)
  rTmp : REAL ;	//Temporary REAL (free for general use)
  dTmp : DINT ;	//Temporary DINT (free for general use)
  UnitNo : INT ;	//Unit Number
  EquipmentID : INT ;	//Equipment ID
  Prid : DINT ;	//Process ID
  SFM36 : STRUCT 	// CIP Pump Mode
   I00 : BOOL ;	// Off
   I01 : BOOL ;	// Flow
   I02 : BOOL ;	// Pressure
   I03 : BOOL ;	// Fix Speed
   I04 : BOOL ;
   I05 : BOOL ;
   I06 : BOOL ;
   I07 : BOOL ;
   I08 : BOOL ;
   I09 : BOOL ;
   I10 : BOOL ;
   I11 : BOOL ;
   I12 : BOOL ;
   I13 : BOOL ;
   I14 : BOOL ;
   I15 : BOOL ;
   I16 : BOOL ;
   I17 : BOOL ;
   I18 : BOOL ;
   I19 : BOOL ;
   I20 : BOOL ;
   I21 : BOOL ;
   I22 : BOOL ;
   I23 : BOOL ;
   I24 : BOOL ;
   I25 : BOOL ;
   I26 : BOOL ;
   I27 : BOOL ;
   I28 : BOOL ;
   I29 : BOOL ;
   I30 : BOOL ;
   I31 : BOOL ;
  END_STRUCT ;
  iPLC : INT ;
  iUnit : INT ;
END_VAR
BEGIN
NETWORK
TITLE =general

      SET   ;

// unit & equipment number ---------------------------------------------------
      L     DB1380.DBW    0;
      T     #UnitNo;

      L     DB1385.DBW   14;
      L     1000;
      *I    ;
      L     #UnitNo;
      +I    ;
      T     #EquipmentID;

// CIP ----------------------------------------------------------------------
      L     DB1385.DBW   18;
      L     0;
      <I    ;
      =     #CIP;

// Communicating Units-------------------------------------------------------
      L     DB1385.DBD   10;
      L     DB1385.DBD  106;
      ==D   ;
      =     #ComCIP;

// emergency OK -------------------------------------------------------------
      A     DB1385.DBX   75.0; //General Emergency Stop OK
      =     #EStopOK;

NETWORK
TITLE =read other unit's data

      SET   ;

// ... General Unit ----------/

      CALL FC   563 (
           ActReq                   := M    101.0,
           PLCNo                    := DB1385.DBW   14,
           SourceUnitNo             := 99,
           IsTUnit                  := FALSE,
           DstComDRec               := DB1385.GEN,
           RET_VAL                  := #wRetVal);


// ... CIP Unit ------------- /

      CALL FC   563 (
           ActReq                   := M    101.0,
           PLCNo                    := 1,
           SourceUnitNo             := 71,
           IsTUnit                  := FALSE,
           DstComDRec               := DB1385.CIP,
           RET_VAL                  := #wRetVal);

//----------------------------------------
// Communication Well Transfer VE1
//----------------------------------------
      L     DB1381.DBD 1134; // Source
      ITD   ;
      DTR   ;
      T     #rTmp;

      CALL FC   950 (
           EquipmentNo              := #rTmp,
           PLCNo                    := #iPLC,
           UnitNo                   := #iUnit);

      CALL FC   563 (
           ActReq                   := M    101.0,
           PLCNo                    := #iPLC,
           SourceUnitNo             := #iUnit,
           IsTUnit                  := FALSE,
           DstComDRec               := DB1385.DST,
           RET_VAL                  := #wRetVal);


NETWORK
TITLE =remote start
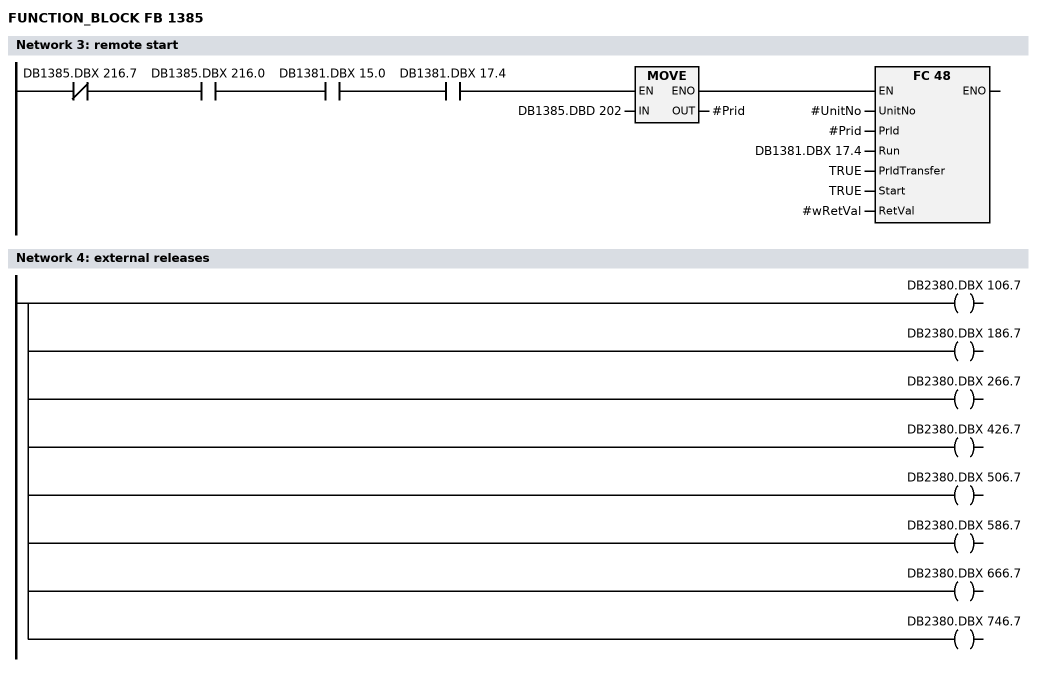

      SET   ;
      AN    DB1385.DBX  216.7;
      A     DB1385.DBX  216.0;
      A     DB1381.DBX   15.0;
      A     DB1381.DBX   17.4;
      JCN   Strt;
      L     DB1385.DBD  202;
      T     #Prid;

      CALL FC    48 (
           UnitNo                   := #UnitNo,
           PrId                     := #Prid,
           Run                      := DB1381.DBX   17.4,
           PrIdTransfer             := TRUE,
           Start                    := TRUE,
           RetVal                   := #wRetVal);
Strt: NOP   0;
NETWORK
TITLE =external releases

      SET   ;
      =     DB2380.DBX  106.7;
      =     DB2380.DBX  186.7;
      =     DB2380.DBX  266.7;
      =     DB2380.DBX  426.7;
      =     DB2380.DBX  506.7;
      =     DB2380.DBX  586.7;
      =     DB2380.DBX  666.7;
      =     DB2380.DBX  746.7;
NETWORK
TITLE =write own unit data

      SET   ;

//-- CIP Communication ---------------------------------------
      AN    DB1381.DBX   15.0;
//      AN "U038SeqD".Seq.PO.B30 // CIP Active (Slave)
      A     #ComCIP;
      JCN   NCIP;
//Conductivity CIP Return
      L     DB1385.DBD  150;
      T     DB1381.DBD  626;

//Temperature CIP Return
      L     DB1385.DBD  146;
      T     DB1381.DBD  594;

//CIP Prerun Pump SP

      CALL FC    45 (
           SFM                      := DB1381.DBD  686,
           Indexes                  := #SFM36);


      L     0.000000e+000;
      A     #SFM36.I01;
      =     DB1385.DBX  171.7;
      JCN   pfc;
      L     DB1381.DBD  654;
pfc:  NOP   0;
      A     #SFM36.I02;
      =     DB1385.DBX  172.0;
      JCN   ppc;
      L     DB1381.DBD  670;
ppc:  NOP   0;
      A     #SFM36.I03;
      =     DB1385.DBX  171.6;
      JCN   pxc;
      L     DB1381.DBD  574;
pxc:  NOP   0;
      T     DB1385.DBD  182;

//CIP Return
      L     DB1381.DBD  558;
      T     DB1385.DBD  186;
      L     DB1385.DBD  138;
      T     DB1381.DBD  562;

//CIP Prerun
      L     DB1381.DBD  542;
      T     DB1385.DBD  190;
      L     DB1385.DBD  142;
      T     DB1381.DBD  546;

// Write Own Data to CIP
      L     DB1385.DBD   10;
      T     DB1385.DBD  154;

      L     DB1385.DBW   14;
      T     DB1385.DBW  158;

      L     DB1385.DBW   16;
      T     DB1385.DBW  160;

      L     DB1385.DBW   18;
      T     DB1385.DBW  162;

      L     DB1385.DBW   20;
      T     DB1385.DBW  164;

      L     DB1385.DBW   22;
      T     DB1385.DBW  166;

      A     DB1385.DBX   24.0;
      =     DB1385.DBX  168.0;

      A     DB1385.DBX   24.1;
      =     DB1385.DBX  168.1;

      A     DB1385.DBX   24.2;
      =     DB1385.DBX  168.2;

      A     DB1385.DBX   24.3;
      =     DB1385.DBX  168.3;

      A     DB1385.DBX   24.4;
      =     DB1385.DBX  168.4;

      A     DB1385.DBX   24.5;
      =     DB1385.DBX  168.5;

      A     DB1385.DBX   24.6;
      =     DB1385.DBX  168.6;

      A     DB1385.DBX   24.7;
      =     DB1385.DBX  168.7;

// Copy Data to CIP
      CALL SFC   20 (
           SRCBLK                   := DB1385.ToCIP,
           RET_VAL                  := #iRetVal,
           DSTBLK                   := DB1385.ToCIP);

NCIP: NOP   0;

//Empty Signal
//A     "U038SpID".SpI.Sig //!!!! Insert correct Empty Signal !!!
      CLR   ;
      =     DB1385.DBX   26.5;

//Full Signal
//A     "U038SpID".SpI.Sig //!!!! Insert correct Full Signal !!!
      CLR   ;
      =     DB1385.DBX   26.2;

//CIP Program Selected
      A     #CIP;
      =     DB1385.DBX   27.1;

// Emergency Stop
      A     #EStopOK; //If needed add or replace with own SpI
      =     DB1385.DBX   27.0; //Emergency Stop OK

// Lifebit
      A     DB2381.DBX  258.7;
      =     DB2380.DBX  748.2;



NETWORK
TITLE = read from other unit data



END_FUNCTION_BLOCK

FUNCTION_BLOCK FB 1389
TITLE =U038: Water Treatment 1
AUTHOR : Woermann
FAMILY : BOTEC_F1
NAME : Sim
VERSION : 0.1


VAR_TEMP
  CIP : BOOL ;	//CIP active
  xTmp : BOOL ;	//Temporary BOOL (free for general use)
  iTmp : INT ;	//Temporary INT (free for general use)
  rTmp : REAL ;	//Temporary REAL (free for general use)
  UnitNo : INT ;	//Unit Number
END_VAR
BEGIN
NETWORK
TITLE =General

      SET   ;
// get unit number ----------------------------------------------------------
      L     DB1380.DBW    0;
      T     #UnitNo;

// CIP ----------------------------------------------------------------------
      L     DB1381.DBD   54;
      L     0;
      <D    ;
      =     #CIP;

NETWORK
TITLE =Actuator

      A     DB1381.DBX   17.3;
      =     DB2380.DBX  105.3;
      =     DB2380.DBX  185.3;
      =     DB2380.DBX  265.3;
      =     DB2380.DBX  425.3;
      =     DB2380.DBX  505.3;
      =     DB2380.DBX  585.3;
      =     DB2380.DBX  665.3;
      =     DB2380.DBX  745.3;

NETWORK
TITLE =Special Input

      A     DB1381.DBX   17.3;
      =     DB2381.DBX   81.3;
      =     DB2381.DBX  141.3;
      =     DB2381.DBX  201.3;
      =     DB2381.DBX  261.3;
      =     DB2381.DBX  321.3;
      =     DB2381.DBX  381.3;
      =     DB2381.DBX  441.3;

NETWORK
TITLE =Counter

      A     DB1381.DBX   17.3;
      A     M    101.0;


      CLR   ;
NETWORK
TITLE =Analog Input

      A     DB1381.DBX   17.3;
      =     DB2383.DBX  141.3;
      =     DB2383.DBX  261.3;
      =     DB2383.DBX  381.3;
      =     DB2383.DBX  501.3;

NETWORK
TITLE =Universal Value

      A     DB1381.DBX   17.3;
//      =     "U038UnVD".unv001.Sim;
//      =     "U038UnVD".unv002.Sim;

NETWORK
TITLE =PID

      A     DB1381.DBX   17.3;

NETWORK
TITLE =Message

      A     DB1381.DBX   17.3;
//      =     "U038MsgD".msg001.Sim;
//      =     "U038MsgD".msg002.Sim;

NETWORK
TITLE =VLT

      A     DB1381.DBX   17.3;

END_FUNCTION_BLOCK

FUNCTION_BLOCK FB 1395
TITLE =U039: Water Treatment 2
FAMILY : BOTEC_F1
NAME : Comm
VERSION : 0.1


VAR_TEMP
  iRetVal : INT ;	//return value as integer
  wRetVal : WORD ;	//return value as word
  Run : BOOL ;	//Unit in "RUN" mode
  EStopOK : BOOL ;	//Emergency Stop OK
  CIP : BOOL ;	//CIP Program Selected
  ComCIP : BOOL ;	//Communication with CIP Active
  xTmp : BOOL ;	//Temporary BOOL (free for general use)
  iTmp : INT ;	//Temporary INT (free for general use)
  rTmp : REAL ;	//Temporary REAL (free for general use)
  dTmp : DINT ;	//Temporary DINT (free for general use)
  UnitNo : INT ;	//Unit Number
  EquipmentID : INT ;	//Equipment ID
  Prid : DINT ;	//Process ID
  SFM36 : STRUCT 	// CIP Pump Mode
   I00 : BOOL ;	// Off
   I01 : BOOL ;	// Flow
   I02 : BOOL ;	// Pressure
   I03 : BOOL ;	// Fix Speed
   I04 : BOOL ;
   I05 : BOOL ;
   I06 : BOOL ;
   I07 : BOOL ;
   I08 : BOOL ;
   I09 : BOOL ;
   I10 : BOOL ;
   I11 : BOOL ;
   I12 : BOOL ;
   I13 : BOOL ;
   I14 : BOOL ;
   I15 : BOOL ;
   I16 : BOOL ;
   I17 : BOOL ;
   I18 : BOOL ;
   I19 : BOOL ;
   I20 : BOOL ;
   I21 : BOOL ;
   I22 : BOOL ;
   I23 : BOOL ;
   I24 : BOOL ;
   I25 : BOOL ;
   I26 : BOOL ;
   I27 : BOOL ;
   I28 : BOOL ;
   I29 : BOOL ;
   I30 : BOOL ;
   I31 : BOOL ;
  END_STRUCT ;
  iPLC : INT ;
  iUnit : INT ;
END_VAR
BEGIN
NETWORK
TITLE =general

      SET   ;

// unit & equipment number ---------------------------------------------------
      L     DB1390.DBW    0;
      T     #UnitNo;

      L     DB1395.DBW   14;
      L     1000;
      *I    ;
      L     #UnitNo;
      +I    ;
      T     #EquipmentID;

// CIP ----------------------------------------------------------------------
      L     DB1395.DBW   18;
      L     0;
      <I    ;
      =     #CIP;

// Communicating Units-------------------------------------------------------
      L     DB1395.DBD   10;
      L     DB1395.DBD  106;
      ==D   ;
      =     #ComCIP;

// emergency OK -------------------------------------------------------------
      A     DB1395.DBX   75.0; //General Emergency Stop OK
      =     #EStopOK;

NETWORK
TITLE =read other unit's data

      SET   ;

// ... General Unit ----------/

      CALL FC   563 (
           ActReq                   := M    101.0,
           PLCNo                    := DB1395.DBW   14,
           SourceUnitNo             := 99,
           IsTUnit                  := FALSE,
           DstComDRec               := DB1395.GEN,
           RET_VAL                  := #wRetVal);


// ... CIP Unit ------------- /

      CALL FC   563 (
           ActReq                   := M    101.0,
           PLCNo                    := 1,
           SourceUnitNo             := 71,
           IsTUnit                  := FALSE,
           DstComDRec               := DB1395.CIP,
           RET_VAL                  := #wRetVal);

//----------------------------------------
// Communication Well Transfer VE2
//----------------------------------------
      L     DB1391.DBD 1134; // Source
      ITD   ;
      DTR   ;
      T     #rTmp;

      CALL FC   950 (
           EquipmentNo              := #rTmp,
           PLCNo                    := #iPLC,
           UnitNo                   := #iUnit);

      CALL FC   563 (
           ActReq                   := M    101.0,
           PLCNo                    := #iPLC,
           SourceUnitNo             := #iUnit,
           IsTUnit                  := FALSE,
           DstComDRec               := DB1395.DST,
           RET_VAL                  := #wRetVal);


NETWORK
TITLE =remote start
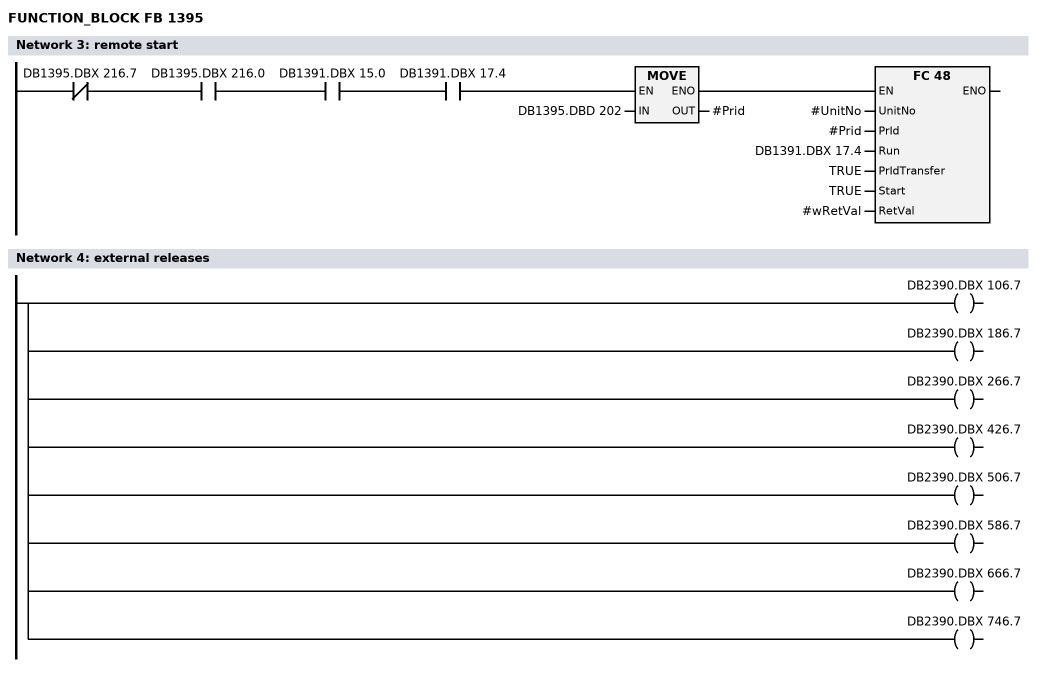

      SET   ;
      AN    DB1395.DBX  216.7;
      A     DB1395.DBX  216.0;
      A     DB1391.DBX   15.0;
      A     DB1391.DBX   17.4;
      JCN   Strt;
      L     DB1395.DBD  202;
      T     #Prid;

      CALL FC    48 (
           UnitNo                   := #UnitNo,
           PrId                     := #Prid,
           Run                      := DB1391.DBX   17.4,
           PrIdTransfer             := TRUE,
           Start                    := TRUE,
           RetVal                   := #wRetVal);
Strt: NOP   0;
NETWORK
TITLE =external releases

      SET   ;
      =     DB2390.DBX  106.7;
      =     DB2390.DBX  186.7;
      =     DB2390.DBX  266.7;
      =     DB2390.DBX  426.7;
      =     DB2390.DBX  506.7;
      =     DB2390.DBX  586.7;
      =     DB2390.DBX  666.7;
      =     DB2390.DBX  746.7;
NETWORK
TITLE =write own unit data

      SET   ;

//-- CIP Communication ---------------------------------------
      AN    DB1391.DBX   15.0;
//      AN "U039SeqD".Seq.PO.B30 // CIP Active (Slave)
      A     #ComCIP;
      JCN   NCIP;
//Conductivity CIP Return
      L     DB1395.DBD  150;
      T     DB1391.DBD  626;

//Temperature CIP Return
      L     DB1395.DBD  146;
      T     DB1391.DBD  594;

//CIP Prerun Pump SP

      CALL FC    45 (
           SFM                      := DB1391.DBD  686,
           Indexes                  := #SFM36);


      L     0.000000e+000;
      A     #SFM36.I01;
      =     DB1395.DBX  171.7;
      JCN   pfc;
      L     DB1391.DBD  654;
pfc:  NOP   0;
      A     #SFM36.I02;
      =     DB1395.DBX  172.0;
      JCN   ppc;
      L     DB1391.DBD  670;
ppc:  NOP   0;
      A     #SFM36.I03;
      =     DB1395.DBX  171.6;
      JCN   pxc;
      L     DB1391.DBD  574;
pxc:  NOP   0;
      T     DB1395.DBD  182;

//CIP Return
      L     DB1391.DBD  558;
      T     DB1395.DBD  186;
      L     DB1395.DBD  138;
      T     DB1391.DBD  562;

//CIP Prerun
      L     DB1391.DBD  542;
      T     DB1395.DBD  190;
      L     DB1395.DBD  142;
      T     DB1391.DBD  546;

// Write Own Data to CIP
      L     DB1395.DBD   10;
      T     DB1395.DBD  154;

      L     DB1395.DBW   14;
      T     DB1395.DBW  158;

      L     DB1395.DBW   16;
      T     DB1395.DBW  160;

      L     DB1395.DBW   18;
      T     DB1395.DBW  162;

      L     DB1395.DBW   20;
      T     DB1395.DBW  164;

      L     DB1395.DBW   22;
      T     DB1395.DBW  166;

      A     DB1395.DBX   24.0;
      =     DB1395.DBX  168.0;

      A     DB1395.DBX   24.1;
      =     DB1395.DBX  168.1;

      A     DB1395.DBX   24.2;
      =     DB1395.DBX  168.2;

      A     DB1395.DBX   24.3;
      =     DB1395.DBX  168.3;

      A     DB1395.DBX   24.4;
      =     DB1395.DBX  168.4;

      A     DB1395.DBX   24.5;
      =     DB1395.DBX  168.5;

      A     DB1395.DBX   24.6;
      =     DB1395.DBX  168.6;

      A     DB1395.DBX   24.7;
      =     DB1395.DBX  168.7;

// Copy Data to CIP
      CALL SFC   20 (
           SRCBLK                   := DB1395.ToCIP,
           RET_VAL                  := #iRetVal,
           DSTBLK                   := DB1395.ToCIP);

NCIP: NOP   0;

//Empty Signal
//A     "U039SpID".SpI.Sig //!!!! Insert correct Empty Signal !!!
      CLR   ;
      =     DB1395.DBX   26.5;

//Full Signal
//A     "U039SpID".SpI.Sig //!!!! Insert correct Full Signal !!!
      CLR   ;
      =     DB1395.DBX   26.2;

//CIP Program Selected
      A     #CIP;
      =     DB1395.DBX   27.1;

// Emergency Stop
      A     #EStopOK; //If needed add or replace with own SpI
      =     DB1395.DBX   27.0; //Emergency Stop OK


// Life bit
      A     DB2391.DBX  258.7;
      =     DB2390.DBX  748.2;


NETWORK
TITLE = read from other unit data



END_FUNCTION_BLOCK

FUNCTION_BLOCK FB 1399
TITLE =U039: Water Treatment 2
AUTHOR : Woermann
FAMILY : BOTEC_F1
NAME : Sim
VERSION : 0.1


VAR_TEMP
  CIP : BOOL ;	//CIP active
  xTmp : BOOL ;	//Temporary BOOL (free for general use)
  iTmp : INT ;	//Temporary INT (free for general use)
  rTmp : REAL ;	//Temporary REAL (free for general use)
  UnitNo : INT ;	//Unit Number
END_VAR
BEGIN
NETWORK
TITLE =General

      SET   ;
// get unit number ----------------------------------------------------------
      L     DB1390.DBW    0;
      T     #UnitNo;

// CIP ----------------------------------------------------------------------
      L     DB1391.DBD   54;
      L     0;
      <D    ;
      =     #CIP;

NETWORK
TITLE =Actuator

      A     DB1391.DBX   17.3;
      =     DB2390.DBX  105.3;
      =     DB2390.DBX  185.3;
      =     DB2390.DBX  265.3;
      =     DB2390.DBX  425.3;
      =     DB2390.DBX  505.3;
      =     DB2390.DBX  585.3;
      =     DB2390.DBX  665.3;
      =     DB2390.DBX  745.3;

NETWORK
TITLE =Special Input

      A     DB1391.DBX   17.3;
      =     DB2391.DBX   81.3;
      =     DB2391.DBX  141.3;
      =     DB2391.DBX  201.3;
      =     DB2391.DBX  261.3;

NETWORK
TITLE =Counter

      A     DB1391.DBX   17.3;
      A     M    101.0;


      CLR   ;
NETWORK
TITLE =Analog Input

      A     DB1391.DBX   17.3;
      =     DB2393.DBX  141.3;
      =     DB2393.DBX  261.3;
      =     DB2393.DBX  381.3;
      =     DB2393.DBX  501.3;

NETWORK
TITLE =Universal Value

      A     DB1391.DBX   17.3;
//      =     "U039UnVD".unv001.Sim;
//      =     "U039UnVD".unv002.Sim;

NETWORK
TITLE =PID

      A     DB1391.DBX   17.3;

NETWORK
TITLE =Message

      A     DB1391.DBX   17.3;
//      =     "U039MsgD".msg001.Sim;
//      =     "U039MsgD".msg002.Sim;

NETWORK
TITLE =VLT

      A     DB1391.DBX   17.3;

END_FUNCTION_BLOCK

FUNCTION_BLOCK FB 1405
TITLE =U040: Water Treatment General
FAMILY : BOTEC_F1
NAME : Comm
VERSION : 0.1


VAR_TEMP
  iRetVal : INT ;	//return value as integer
  wRetVal : WORD ;	//return value as word
  Run : BOOL ;	//Unit in "RUN" mode
  EStopOK : BOOL ;	//Emergency Stop OK
  CIP : BOOL ;	//CIP Program Selected
  ComCIP : BOOL ;	//Communication with CIP Active
  xTmp : BOOL ;	//Temporary BOOL (free for general use)
  iTmp : INT ;	//Temporary INT (free for general use)
  rTmp : REAL ;	//Temporary REAL (free for general use)
  dTmp : DINT ;	//Temporary DINT (free for general use)
  UnitNo : INT ;	//Unit Number
  EquipmentID : INT ;	//Equipment ID
  Prid : DINT ;	//Process ID
  SFM36 : STRUCT 	// CIP Pump Mode
   I00 : BOOL ;	// Off
   I01 : BOOL ;	// Flow
   I02 : BOOL ;	// Pressure
   I03 : BOOL ;	// Fix Speed
   I04 : BOOL ;
   I05 : BOOL ;
   I06 : BOOL ;
   I07 : BOOL ;
   I08 : BOOL ;
   I09 : BOOL ;
   I10 : BOOL ;
   I11 : BOOL ;
   I12 : BOOL ;
   I13 : BOOL ;
   I14 : BOOL ;
   I15 : BOOL ;
   I16 : BOOL ;
   I17 : BOOL ;
   I18 : BOOL ;
   I19 : BOOL ;
   I20 : BOOL ;
   I21 : BOOL ;
   I22 : BOOL ;
   I23 : BOOL ;
   I24 : BOOL ;
   I25 : BOOL ;
   I26 : BOOL ;
   I27 : BOOL ;
   I28 : BOOL ;
   I29 : BOOL ;
   I30 : BOOL ;
   I31 : BOOL ;
  END_STRUCT ;
END_VAR
BEGIN
NETWORK
TITLE =general

      SET   ;

